KUKA KRL program: ps_604c1.src, ps_604c1.dat

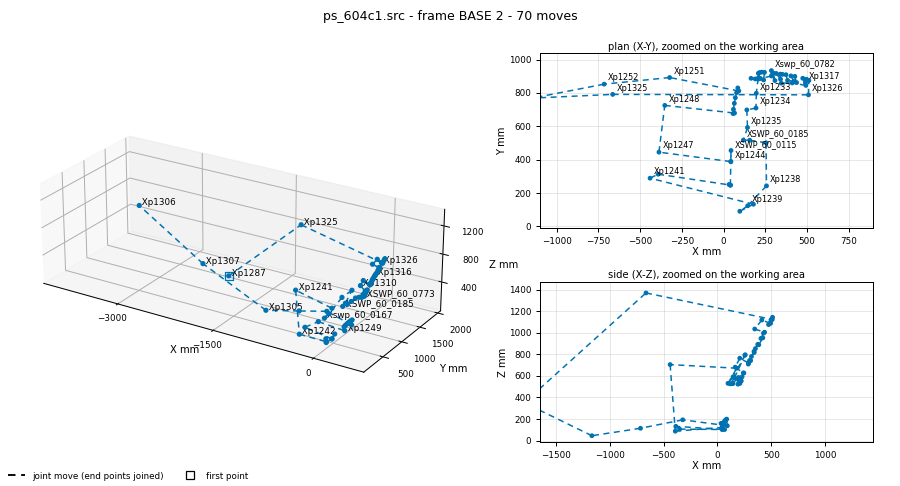
[picture p0: tool path of ps_604c1.src in frame BASE 2, 70 of 70 moves have a stored position in this frame; points joined in program order, loops and branches not executed]
--- ps_604c1.src ---
&ACCESS RVO2
&REL 166
&COMMENT Geom C1 Accelo Atual sem o PTO 60-0682
DEF ps_604c1( )
EXT e_Fraes1 ( )
EXT f_Fraes1 ( )
  ;FOLD INI;%{PE}%V2.2.2,%MKUKATPBASIS,%CINIT,%VCOMMON,%P
  ;FOLD BAS INI;%{PE}%V2.2.2,%MKUKATPBASIS,%CINIT,%VINIT,%P
  INTERRUPT DECL 3 WHEN $STOPMESS==TRUE DO IR_STOPM ( )
  INTERRUPT ON 3
  BAS (#INITMOV,0 )
  ;ENDFOLD
  ;FOLD A20 INI;%{E}%V2.2.2,%MKUKATPA20,%CINIT,%VINIT,%P
  IF ARC20==TRUE THEN
    A20 (ARC_INI)
    INTERRUPT DECL 6 WHEN $CYCFLAG[3]==FALSE DO A20(TECH_STOP2)
  ENDIF
  ;ENDFOLD
  ;FOLD A10 INI;%{E}%V2.2.2,%MKUKATPARC,%CINIT,%VINIT,%P
  IF A10_OPTION==#ACTIVE THEN
    INTERRUPT DECL 4 WHEN $CYCFLAG[2]==FALSE DO A10 (#APPL_ERROR)
    INTERRUPT DECL 7 WHEN A_ARC_SWI==#ACTIVE DO A10 (#ARC_SEAM)
    INTERRUPT DECL 5 WHEN A_FLY_ARC==TRUE DO A10 (#HPU_ARC)
    INTERRUPT  ON 5
    A10_INI ( )
  ENDIF
  ;ENDFOLD
  ;FOLD GRIPPER INI;%{E}%V2.2.2,%MKUKATPGRIPPER,%CINIT,%VINIT,%P
  USER_GRP(0,DUMMY,DUMMY,GDEFAULT)
  ;ENDFOLD
  ;FOLD SPOT INI;%{E}%V.2.2,%MKUKATPSPOT,%CINIT,%VINIT,%P
  USERSPOT(#INIT)
  ;ENDFOLD
  ;FOLD TOUCHSENSE INI;%{E}%V2.2.2,%MKUKATPTS,%CINIT,%VINIT,%P
  IF H70_OPTION THEN
    INTERRUPT DECL 15 WHEN $MEAS_PULSE[TOUCH_I[TOUCH_ACTIVE].IN_NR] DO H70 (6,CD0 )
    INTERRUPT DECL 16 WHEN $ZERO_MOVE DO H70 (7,CD0 )
    INTERRUPT DECL 17 WHEN $TECHPAR_C[FG_TOUCH,8]>0.5 DO H70 (8,CD0)
    H70 (1,CD0 )
  ENDIF
  ;ENDFOLD
  ;FOLD USER INI;%{P}%V2.2.2,%MKUKATPUSER,%CINIT,%VINIT,%P
  ;Make your modifications here
  ;ENDFOLD
  ;ENDFOLD

; Caracterização dos meios de produção: P13.060-R4
; Versão atual: 20/07/2013 12:00  Nome: Solda Geometria C1
; Change: Accelo

chk_w1_wechs_ok ( )     ; VERIFICAÇÃO DE FERRAMENTA: C1

;FOLD PTP p1287 CONT Vel= 80 % PDAT118 Tool[1]:GUN C1 Base[2]:Accelo;%{PE}%R 4.1.16,%MKUKATPBASIS,%CMOVE,%VPTP,%P 1:PTP, 2:p1287, 3:C_PTP, 5:80, 7:PDAT118
$BWDSTART = FALSE
PDAT_ACT=PPDAT118
BAS(#PTP_DAT)
FDAT_ACT=Fp1287
BAS(#FRAMES)
BAS(#VEL_PTP,80)
PTP Xp1287 C_PTP
;ENDFOLD

;FOLD OUT 848 'Area de Solda'  State= FALSE ;%{PE}%R 4.1.16,%MKUKATPBASIS,%COUT,%VOUTX,%P 2:848, 3:'Area de Solda', 5:FALSE, 6:
$OUT[848]=FALSE
;ENDFOLD

;FOLD PTP p1325 CONT Vel= 80 % PDAT36 Tool[1]:GUN C1 Base[2]:Accelo;%{PE}%R 4.1.16,%MKUKATPBASIS,%CMOVE,%VPTP,%P 1:PTP, 2:p1325, 3:C_PTP, 5:80, 7:PDAT36
$BWDSTART = FALSE
PDAT_ACT=PPDAT36
BAS(#PTP_DAT)
FDAT_ACT=Fp1325
BAS(#FRAMES)
BAS(#VEL_PTP,80)
PTP Xp1325 C_PTP
;ENDFOLD
;FOLD PTP p1326 CONT Vel= 80 % PDAT37 Tool[1]:GUN C1 Base[2]:Accelo;%{PE}%R 4.1.16,%MKUKATPBASIS,%CMOVE,%VPTP,%P 1:PTP, 2:p1326, 3:C_PTP, 5:80, 7:PDAT37
$BWDSTART = FALSE
PDAT_ACT=PPDAT37
BAS(#PTP_DAT)
FDAT_ACT=Fp1326
BAS(#FRAMES)
BAS(#VEL_PTP,80)
PTP Xp1326 C_PTP
;ENDFOLD


;FOLD OUT 839 'R4 Soldando'  State= TRUE ;%{PE}%R 4.1.16,%MKUKATPBASIS,%COUT,%VOUTX,%P 2:839, 3:'R4 Soldando', 5:TRUE, 6:
$OUT[839]=TRUE
;ENDFOLD

;FOLD ;  SWP_60_0806;%{PE}%R 4.1.16,%MKUKATPBASIS,%CCOMMENT,%VNORMAL,%P 2: SWP_60_0806
;ENDFOLD
;FOLD PTP swp_60_0806 PDAT38 SPOT Gun= 1 RETR OPN PgNo1= 16 ACTIVE= 1 Tool[1]:GUN C1 Base[2]:Accelo;%{PE}%R 4.1.12,%MKUKATPSPOT,%CSPOT,%VPTP,%P 1:PTP, 2:swp_60_0806, 3:, 5:100, 7:PDAT38, 10:1, 12:#FIRST, 14:#OPN, 16:16, 18:1, 20:0, 22:0, 24:1, 25:NORMAL8
$BWDSTART = FALSE
PDAT_ACT=PPDAT38
BAS(#PTP_DAT)
FDAT_ACT=Fswp_60_0806
BAS(#FRAMES)
BAS(#VEL_PTP,PPDAT38.VEL)
S_ACT.GUN=1
S_ACT.PAIR=SDEFAULT.PAIR
S_ACT.RETR=#OPN
S_ACT.CLO_TM=1
S_ACT.PGNO1=16
S_ACT.PGNO2=SDEFAULT.PGNO2
S_ACT.PRESS1=SDEFAULT.PRESS1
S_ACT.PRESS2=SDEFAULT.PRESS2
S_READY=FALSE
PTP Xswp_60_0806
USERSPOT(#SPOT, S_ACT)
WAIT FOR S_READY
;ENDFOLD

;FOLD ;  SWP_60_0804;%{PE}%R 4.1.16,%MKUKATPBASIS,%CCOMMENT,%VNORMAL,%P 2: SWP_60_0804
;ENDFOLD
;FOLD PTP swp_60_0804 PDAT39 SPOT Gun= 1 RETR OPN PgNo1= 17 ACTIVE= 1 Tool[1]:GUN C1 Base[2]:Accelo;%{PE}%R 4.1.12,%MKUKATPSPOT,%CSPOT,%VPTP,%P 1:PTP, 2:swp_60_0804, 3:, 5:100, 7:PDAT39, 10:1, 12:#FIRST, 14:#OPN, 16:17, 18:1, 20:0, 22:0, 24:1, 25:NORMAL9
$BWDSTART = FALSE
PDAT_ACT=PPDAT39
BAS(#PTP_DAT)
FDAT_ACT=Fswp_60_0804
BAS(#FRAMES)
BAS(#VEL_PTP,PPDAT39.VEL)
S_ACT.GUN=1
S_ACT.PAIR=SDEFAULT.PAIR
S_ACT.RETR=#OPN
S_ACT.CLO_TM=1
S_ACT.PGNO1=17
S_ACT.PGNO2=SDEFAULT.PGNO2
S_ACT.PRESS1=SDEFAULT.PRESS1
S_ACT.PRESS2=SDEFAULT.PRESS2
S_READY=FALSE
PTP Xswp_60_0804
USERSPOT(#SPOT, S_ACT)
WAIT FOR S_READY
;ENDFOLD

;FOLD PTP p1317 CONT Vel= 70 % PDAT40 Tool[1]:GUN C1 Base[2]:Accelo;%{PE}%R 4.1.16,%MKUKATPBASIS,%CMOVE,%VPTP,%P 1:PTP, 2:p1317, 3:C_PTP, 5:70, 7:PDAT40
$BWDSTART = FALSE
PDAT_ACT=PPDAT40
BAS(#PTP_DAT)
FDAT_ACT=Fp1317
BAS(#FRAMES)
BAS(#VEL_PTP,70)
PTP Xp1317 C_PTP
;ENDFOLD

;FOLD ;  SWP_60_0802;%{PE}%R 4.1.16,%MKUKATPBASIS,%CCOMMENT,%VNORMAL,%P 2: SWP_60_0802
;ENDFOLD
;FOLD PTP swp_60_0802 PDAT41 SPOT Gun= 1 RETR OPN PgNo1= 18 ACTIVE= 1 Tool[1]:GUN C1 Base[2]:Accelo;%{PE}%R 4.1.12,%MKUKATPSPOT,%CSPOT,%VPTP,%P 1:PTP, 2:swp_60_0802, 3:, 5:100, 7:PDAT41, 10:1, 12:#FIRST, 14:#OPN, 16:18, 18:1, 20:0, 22:0, 24:1, 25:NORMAL10
$BWDSTART = FALSE
PDAT_ACT=PPDAT41
BAS(#PTP_DAT)
FDAT_ACT=Fswp_60_0802
BAS(#FRAMES)
BAS(#VEL_PTP,PPDAT41.VEL)
S_ACT.GUN=1
S_ACT.PAIR=SDEFAULT.PAIR
S_ACT.RETR=#OPN
S_ACT.CLO_TM=1
S_ACT.PGNO1=18
S_ACT.PGNO2=SDEFAULT.PGNO2
S_ACT.PRESS1=SDEFAULT.PRESS1
S_ACT.PRESS2=SDEFAULT.PRESS2
S_READY=FALSE
PTP Xswp_60_0802
USERSPOT(#SPOT, S_ACT)
WAIT FOR S_READY
;ENDFOLD

;FOLD PTP p1226 CONT Vel= 100 % PDAT57 Tool[1]:GUN C1 Base[2]:Accelo;%{PE}%R 4.1.16,%MKUKATPBASIS,%CMOVE,%VPTP,%P 1:PTP, 2:p1226, 3:C_PTP, 5:100, 7:PDAT57
$BWDSTART = FALSE
PDAT_ACT=PPDAT57
BAS(#PTP_DAT)
FDAT_ACT=Fp1226
BAS(#FRAMES)
BAS(#VEL_PTP,100)
PTP Xp1226 C_PTP
;ENDFOLD
;FOLD PTP p1227 CONT Vel= 100 % PDAT58 Tool[1]:GUN C1 Base[2]:Accelo;%{PE}%R 4.1.16,%MKUKATPBASIS,%CMOVE,%VPTP,%P 1:PTP, 2:p1227, 3:C_PTP, 5:100, 7:PDAT58
$BWDSTART = FALSE
PDAT_ACT=PPDAT58
BAS(#PTP_DAT)
FDAT_ACT=Fp1227
BAS(#FRAMES)
BAS(#VEL_PTP,100)
PTP Xp1227 C_PTP
;ENDFOLD
;FOLD PTP p1228 CONT Vel= 100 % PDAT59 Tool[1]:GUN C1 Base[2]:Accelo;%{PE}%R 4.1.16,%MKUKATPBASIS,%CMOVE,%VPTP,%P 1:PTP, 2:p1228, 3:C_PTP, 5:100, 7:PDAT59
$BWDSTART = FALSE
PDAT_ACT=PPDAT59
BAS(#PTP_DAT)
FDAT_ACT=Fp1228
BAS(#FRAMES)
BAS(#VEL_PTP,100)
PTP Xp1228 C_PTP
;ENDFOLD
;FOLD PTP p1229 CONT Vel= 100 % PDAT60 Tool[1]:GUN C1 Base[2]:Accelo;%{PE}%R 4.1.16,%MKUKATPBASIS,%CMOVE,%VPTP,%P 1:PTP, 2:p1229, 3:C_PTP, 5:100, 7:PDAT60
$BWDSTART = FALSE
PDAT_ACT=PPDAT60
BAS(#PTP_DAT)
FDAT_ACT=Fp1229
BAS(#FRAMES)
BAS(#VEL_PTP,100)
PTP Xp1229 C_PTP
;ENDFOLD

;FOLD ;  SWP_60_0798;%{PE}%R 4.1.16,%MKUKATPBASIS,%CCOMMENT,%VNORMAL,%P 2: SWP_60_0798
;ENDFOLD
;FOLD PTP swp_60_0798 PDAT43 SPOT Gun= 1 RETR OPN PgNo1= 20 ACTIVE= 1 Tool[1]:GUN C1 Base[2]:Accelo;%{PE}%R 4.1.12,%MKUKATPSPOT,%CSPOT,%VPTP,%P 1:PTP, 2:swp_60_0798, 3:, 5:100, 7:PDAT43, 10:1, 12:#FIRST, 14:#OPN, 16:20, 18:1, 20:0, 22:0, 24:1, 25:NORMAL12
$BWDSTART = FALSE
PDAT_ACT=PPDAT43
BAS(#PTP_DAT)
FDAT_ACT=Fswp_60_0798
BAS(#FRAMES)
BAS(#VEL_PTP,PPDAT43.VEL)
S_ACT.GUN=1
S_ACT.PAIR=SDEFAULT.PAIR
S_ACT.RETR=#OPN
S_ACT.CLO_TM=1
S_ACT.PGNO1=20
S_ACT.PGNO2=SDEFAULT.PGNO2
S_ACT.PRESS1=SDEFAULT.PRESS1
S_ACT.PRESS2=SDEFAULT.PRESS2
S_READY=FALSE
PTP Xswp_60_0798
USERSPOT(#SPOT, S_ACT)
WAIT FOR S_READY
;ENDFOLD

;FOLD ;  SWP_60_0794;%{PE}%R 4.1.16,%MKUKATPBASIS,%CCOMMENT,%VNORMAL,%P 2: SWP_60_0794
;ENDFOLD
;FOLD PTP swp_60_0794 PDAT44 SPOT Gun= 1 RETR OPN PgNo1= 21 ACTIVE= 1 Tool[1]:GUN C1 Base[2]:Accelo;%{PE}%R 4.1.12,%MKUKATPSPOT,%CSPOT,%VPTP,%P 1:PTP, 2:swp_60_0794, 3:, 5:100, 7:PDAT44, 10:1, 12:#FIRST, 14:#OPN, 16:21, 18:1, 20:0, 22:0, 24:1, 25:NORMAL13
$BWDSTART = FALSE
PDAT_ACT=PPDAT44
BAS(#PTP_DAT)
FDAT_ACT=Fswp_60_0794
BAS(#FRAMES)
BAS(#VEL_PTP,PPDAT44.VEL)
S_ACT.GUN=1
S_ACT.PAIR=SDEFAULT.PAIR
S_ACT.RETR=#OPN
S_ACT.CLO_TM=1
S_ACT.PGNO1=21
S_ACT.PGNO2=SDEFAULT.PGNO2
S_ACT.PRESS1=SDEFAULT.PRESS1
S_ACT.PRESS2=SDEFAULT.PRESS2
S_READY=FALSE
PTP Xswp_60_0794
USERSPOT(#SPOT, S_ACT)
WAIT FOR S_READY
;ENDFOLD

;FOLD PTP p1282 CONT Vel= 80 % P_OLP77 Tool[1]:GUN C1 Base[2]:Accelo;%{PE}%R 4.1.16,%MKUKATPBASIS,%CMOVE,%VPTP,%P 1:PTP, 2:p1282, 3:C_PTP, 5:80, 7:P_OLP77
$BWDSTART = FALSE
PDAT_ACT=PP_OLP77
BAS(#PTP_DAT)
FDAT_ACT=Fp1282
BAS(#FRAMES)
BAS(#VEL_PTP,80)
PTP Xp1282 C_PTP
;ENDFOLD
;FOLD PTP p1316 CONT Vel= 80 % PDAT45 Tool[1]:GUN C1 Base[2]:Accelo;%{PE}%R 4.1.16,%MKUKATPBASIS,%CMOVE,%VPTP,%P 1:PTP, 2:p1316, 3:C_PTP, 5:80, 7:PDAT45
$BWDSTART = FALSE
PDAT_ACT=PPDAT45
BAS(#PTP_DAT)
FDAT_ACT=Fp1316
BAS(#FRAMES)
BAS(#VEL_PTP,80)
PTP Xp1316 C_PTP
;ENDFOLD

;FOLD ;  SWP_60_0792;%{PE}%R 4.1.16,%MKUKATPBASIS,%CCOMMENT,%VNORMAL,%P 2: SWP_60_0792
;ENDFOLD
;FOLD PTP swp_60_0792 PDAT46 SPOT Gun= 1 RETR OPN PgNo1= 22 ACTIVE= 1 Tool[1]:GUN C1 Base[2]:Accelo;%{PE}%R 4.1.12,%MKUKATPSPOT,%CSPOT,%VPTP,%P 1:PTP, 2:swp_60_0792, 3:, 5:100, 7:PDAT46, 10:1, 12:#FIRST, 14:#OPN, 16:22, 18:1, 20:0, 22:0, 24:1, 25:NORMAL14
$BWDSTART = FALSE
PDAT_ACT=PPDAT46
BAS(#PTP_DAT)
FDAT_ACT=Fswp_60_0792
BAS(#FRAMES)
BAS(#VEL_PTP,PPDAT46.VEL)
S_ACT.GUN=1
S_ACT.PAIR=SDEFAULT.PAIR
S_ACT.RETR=#OPN
S_ACT.CLO_TM=1
S_ACT.PGNO1=22
S_ACT.PGNO2=SDEFAULT.PGNO2
S_ACT.PRESS1=SDEFAULT.PRESS1
S_ACT.PRESS2=SDEFAULT.PRESS2
S_READY=FALSE
PTP Xswp_60_0792
USERSPOT(#SPOT, S_ACT)
WAIT FOR S_READY
;ENDFOLD

;FOLD ;  SWP_60_0790;%{PE}%R 4.1.16,%MKUKATPBASIS,%CCOMMENT,%VNORMAL,%P 2: SWP_60_0790
;ENDFOLD
;FOLD PTP swp_60_0790 PDAT47 SPOT Gun= 1 RETR OPN PgNo1= 23 ACTIVE= 1 Tool[1]:GUN C1 Base[2]:Accelo;%{PE}%R 4.1.12,%MKUKATPSPOT,%CSPOT,%VPTP,%P 1:PTP, 2:swp_60_0790, 3:, 5:100, 7:PDAT47, 10:1, 12:#FIRST, 14:#OPN, 16:23, 18:1, 20:0, 22:0, 24:1, 25:NORMAL15
$BWDSTART = FALSE
PDAT_ACT=PPDAT47
BAS(#PTP_DAT)
FDAT_ACT=Fswp_60_0790
BAS(#FRAMES)
BAS(#VEL_PTP,PPDAT47.VEL)
S_ACT.GUN=1
S_ACT.PAIR=SDEFAULT.PAIR
S_ACT.RETR=#OPN
S_ACT.CLO_TM=1
S_ACT.PGNO1=23
S_ACT.PGNO2=SDEFAULT.PGNO2
S_ACT.PRESS1=SDEFAULT.PRESS1
S_ACT.PRESS2=SDEFAULT.PRESS2
S_READY=FALSE
PTP Xswp_60_0790
USERSPOT(#SPOT, S_ACT)
WAIT FOR S_READY
;ENDFOLD

;FOLD ;  SWP_60_0788;%{PE}%R 4.1.16,%MKUKATPBASIS,%CCOMMENT,%VNORMAL,%P 2: SWP_60_0788
;ENDFOLD
;FOLD PTP swp_60_0788 PDAT48 SPOT Gun= 1 RETR OPN PgNo1= 24 ACTIVE= 1 Tool[1]:GUN C1 Base[2]:Accelo;%{PE}%R 4.1.12,%MKUKATPSPOT,%CSPOT,%VPTP,%P 1:PTP, 2:swp_60_0788, 3:, 5:100, 7:PDAT48, 10:1, 12:#FIRST, 14:#OPN, 16:24, 18:1, 20:0, 22:0, 24:1, 25:NORMAL16
$BWDSTART = FALSE
PDAT_ACT=PPDAT48
BAS(#PTP_DAT)
FDAT_ACT=Fswp_60_0788
BAS(#FRAMES)
BAS(#VEL_PTP,PPDAT48.VEL)
S_ACT.GUN=1
S_ACT.PAIR=SDEFAULT.PAIR
S_ACT.RETR=#OPN
S_ACT.CLO_TM=1
S_ACT.PGNO1=24
S_ACT.PGNO2=SDEFAULT.PGNO2
S_ACT.PRESS1=SDEFAULT.PRESS1
S_ACT.PRESS2=SDEFAULT.PRESS2
S_READY=FALSE
PTP Xswp_60_0788
USERSPOT(#SPOT, S_ACT)
WAIT FOR S_READY
;ENDFOLD

;FOLD PTP p1321 CONT Vel= 80 % PDAT49 Tool[1]:GUN C1 Base[2]:Accelo;%{PE}%R 4.1.16,%MKUKATPBASIS,%CMOVE,%VPTP,%P 1:PTP, 2:p1321, 3:C_PTP, 5:80, 7:PDAT49
$BWDSTART = FALSE
PDAT_ACT=PPDAT49
BAS(#PTP_DAT)
FDAT_ACT=Fp1321
BAS(#FRAMES)
BAS(#VEL_PTP,80)
PTP Xp1321 C_PTP
;ENDFOLD

;FOLD ;  SWP_60_0786;%{PE}%R 4.1.16,%MKUKATPBASIS,%CCOMMENT,%VNORMAL,%P 2: SWP_60_0786
;ENDFOLD
;FOLD PTP swp_60_0786 PDAT50 SPOT Gun= 1 RETR OPN PgNo1= 25 ACTIVE= 1 Tool[1]:GUN C1 Base[2]:Accelo;%{PE}%R 4.1.12,%MKUKATPSPOT,%CSPOT,%VPTP,%P 1:PTP, 2:swp_60_0786, 3:, 5:100, 7:PDAT50, 10:1, 12:#FIRST, 14:#OPN, 16:25, 18:1, 20:0, 22:0, 24:1, 25:NORMAL17
$BWDSTART = FALSE
PDAT_ACT=PPDAT50
BAS(#PTP_DAT)
FDAT_ACT=Fswp_60_0786
BAS(#FRAMES)
BAS(#VEL_PTP,PPDAT50.VEL)
S_ACT.GUN=1
S_ACT.PAIR=SDEFAULT.PAIR
S_ACT.RETR=#OPN
S_ACT.CLO_TM=1
S_ACT.PGNO1=25
S_ACT.PGNO2=SDEFAULT.PGNO2
S_ACT.PRESS1=SDEFAULT.PRESS1
S_ACT.PRESS2=SDEFAULT.PRESS2
S_READY=FALSE
PTP Xswp_60_0786
USERSPOT(#SPOT, S_ACT)
WAIT FOR S_READY
;ENDFOLD

;FOLD ;  SWP_60_0784;%{PE}%R 4.1.16,%MKUKATPBASIS,%CCOMMENT,%VNORMAL,%P 2: SWP_60_0784
;ENDFOLD
;FOLD PTP SWP_60_0785 PDAT117 SPOT Gun= 1 RETR OPN PgNo1= 5 ACTIVE= 1 Tool[1]:GUN C1 Base[2]:Accelo;%{PE}%R 4.1.12,%MKUKATPSPOT,%CSPOT,%VPTP,%P 1:PTP, 2:SWP_60_0785, 3:, 5:100, 7:PDAT117, 10:1, 12:#FIRST, 14:#OPN, 16:5, 18:1, 20:0, 22:0, 24:1, 25:NORMAL22
$BWDSTART = FALSE
PDAT_ACT=PPDAT117
BAS(#PTP_DAT)
FDAT_ACT=FSWP_60_0785
BAS(#FRAMES)
BAS(#VEL_PTP,PPDAT117.VEL)
S_ACT.GUN=1
S_ACT.PAIR=SDEFAULT.PAIR
S_ACT.RETR=#OPN
S_ACT.CLO_TM=1
S_ACT.PGNO1=5
S_ACT.PGNO2=SDEFAULT.PGNO2
S_ACT.PRESS1=SDEFAULT.PRESS1
S_ACT.PRESS2=SDEFAULT.PRESS2
S_READY=FALSE
PTP XSWP_60_0785
USERSPOT(#SPOT, S_ACT)
WAIT FOR S_READY
;ENDFOLD

;FOLD PTP p1322 CONT Vel= 100 % PDAT51 Tool[1]:GUN C1 Base[2]:Accelo;%{PE}%R 4.1.16,%MKUKATPBASIS,%CMOVE,%VPTP,%P 1:PTP, 2:p1322, 3:C_PTP, 5:100, 7:PDAT51
$BWDSTART = FALSE
PDAT_ACT=PPDAT51
BAS(#PTP_DAT)
FDAT_ACT=Fp1322
BAS(#FRAMES)
BAS(#VEL_PTP,100)
PTP Xp1322 C_PTP
;ENDFOLD
;FOLD PTP p1323 CONT Vel= 100 % PDAT52 Tool[1]:GUN C1 Base[2]:Accelo;%{PE}%R 4.1.16,%MKUKATPBASIS,%CMOVE,%VPTP,%P 1:PTP, 2:p1323, 3:C_PTP, 5:100, 7:PDAT52
$BWDSTART = FALSE
PDAT_ACT=PPDAT52
BAS(#PTP_DAT)
FDAT_ACT=Fp1323
BAS(#FRAMES)
BAS(#VEL_PTP,100)
PTP Xp1323 C_PTP
;ENDFOLD

;FOLD ;  SWP_60_0782;%{PE}%R 4.1.16,%MKUKATPBASIS,%CCOMMENT,%VNORMAL,%P 2: SWP_60_0782
;ENDFOLD
;FOLD PTP swp_60_0782 PDAT53 SPOT Gun= 1 RETR OPN PgNo1= 26 ACTIVE= 1 Tool[1]:GUN C1 Base[2]:Accelo;%{PE}%R 4.1.12,%MKUKATPSPOT,%CSPOT,%VPTP,%P 1:PTP, 2:swp_60_0782, 3:, 5:100, 7:PDAT53, 10:1, 12:#FIRST, 14:#OPN, 16:26, 18:1, 20:0, 22:0, 24:1, 25:NORMAL18
$BWDSTART = FALSE
PDAT_ACT=PPDAT53
BAS(#PTP_DAT)
FDAT_ACT=Fswp_60_0782
BAS(#FRAMES)
BAS(#VEL_PTP,PPDAT53.VEL)
S_ACT.GUN=1
S_ACT.PAIR=SDEFAULT.PAIR
S_ACT.RETR=#OPN
S_ACT.CLO_TM=1
S_ACT.PGNO1=26
S_ACT.PGNO2=SDEFAULT.PGNO2
S_ACT.PRESS1=SDEFAULT.PRESS1
S_ACT.PRESS2=SDEFAULT.PRESS2
S_READY=FALSE
PTP Xswp_60_0782
USERSPOT(#SPOT, S_ACT)
WAIT FOR S_READY
;ENDFOLD

;FOLD PTP p1327 CONT Vel= 80 % PDAT55 Tool[1]:GUN C1 Base[2]:Accelo;%{PE}%R 4.1.16,%MKUKATPBASIS,%CMOVE,%VPTP,%P 1:PTP, 2:p1327, 3:C_PTP, 5:80, 7:PDAT55
$BWDSTART = FALSE
PDAT_ACT=PPDAT55
BAS(#PTP_DAT)
FDAT_ACT=Fp1327
BAS(#FRAMES)
BAS(#VEL_PTP,80)
PTP Xp1327 C_PTP
;ENDFOLD
;FOLD PTP p1328 CONT Vel= 80 % PDAT56 Tool[1]:GUN C1 Base[2]:Accelo;%{PE}%R 4.1.16,%MKUKATPBASIS,%CMOVE,%VPTP,%P 1:PTP, 2:p1328, 3:C_PTP, 5:80, 7:PDAT56
$BWDSTART = FALSE
PDAT_ACT=PPDAT56
BAS(#PTP_DAT)
FDAT_ACT=Fp1328
BAS(#FRAMES)
BAS(#VEL_PTP,80)
PTP Xp1328 C_PTP
;ENDFOLD
;FOLD PTP p1310 CONT Vel= 90 % P_OLP78 Tool[1]:GUN C1 Base[2]:Accelo;%{PE}%R 4.1.16,%MKUKATPBASIS,%CMOVE,%VPTP,%P 1:PTP, 2:p1310, 3:C_PTP, 5:90, 7:P_OLP78
$BWDSTART = FALSE
PDAT_ACT=PP_OLP78
BAS(#PTP_DAT)
FDAT_ACT=Fp1310
BAS(#FRAMES)
BAS(#VEL_PTP,90)
PTP Xp1310 C_PTP
;ENDFOLD
;FOLD PTP p1231 CONT Vel= 80 % PDAT62 Tool[1]:GUN C1 Base[2]:Accelo;%{PE}%R 4.1.16,%MKUKATPBASIS,%CMOVE,%VPTP,%P 1:PTP, 2:p1231, 3:C_PTP, 5:80, 7:PDAT62
$BWDSTART = FALSE
PDAT_ACT=PPDAT62
BAS(#PTP_DAT)
FDAT_ACT=Fp1231
BAS(#FRAMES)
BAS(#VEL_PTP,80)
PTP Xp1231 C_PTP
;ENDFOLD

;FOLD ;  SWP_60_0778;%{PE}%R 4.1.16,%MKUKATPBASIS,%CCOMMENT,%VNORMAL,%P 2: SWP_60_0778
;ENDFOLD
;FOLD PTP swp_60_0779 PDAT63 SPOT Gun= 1 RETR OPN PgNo1= 28 ACTIVE= 1 Tool[1]:GUN C1 Base[2]:Accelo;%{PE}%R 4.1.12,%MKUKATPSPOT,%CSPOT,%VPTP,%P 1:PTP, 2:swp_60_0779, 3:, 5:100, 7:PDAT63, 10:1, 12:#FIRST, 14:#OPN, 16:28, 18:1, 20:0, 22:0, 24:1, 25:NORMAL20
$BWDSTART = FALSE
PDAT_ACT=PPDAT63
BAS(#PTP_DAT)
FDAT_ACT=Fswp_60_0779
BAS(#FRAMES)
BAS(#VEL_PTP,PPDAT63.VEL)
S_ACT.GUN=1
S_ACT.PAIR=SDEFAULT.PAIR
S_ACT.RETR=#OPN
S_ACT.CLO_TM=1
S_ACT.PGNO1=28
S_ACT.PGNO2=SDEFAULT.PGNO2
S_ACT.PRESS1=SDEFAULT.PRESS1
S_ACT.PRESS2=SDEFAULT.PRESS2
S_READY=FALSE
PTP Xswp_60_0779
USERSPOT(#SPOT, S_ACT)
WAIT FOR S_READY
;ENDFOLD

;FOLD ;  SWP_60_0776;%{PE}%R 4.1.16,%MKUKATPBASIS,%CCOMMENT,%VNORMAL,%P 2: SWP_60_0776
;ENDFOLD
;FOLD PTP swp_60_0777 PDAT64 SPOT Gun= 1 RETR OPN PgNo1= 29 ACTIVE= 1 Tool[1]:GUN C1 Base[2]:Accelo;%{PE}%R 4.1.12,%MKUKATPSPOT,%CSPOT,%VPTP,%P 1:PTP, 2:swp_60_0777, 3:, 5:100, 7:PDAT64, 10:1, 12:#FIRST, 14:#OPN, 16:29, 18:1, 20:0, 22:0, 24:1, 25:NORMAL20
$BWDSTART = FALSE
PDAT_ACT=PPDAT64
BAS(#PTP_DAT)
FDAT_ACT=Fswp_60_0777
BAS(#FRAMES)
BAS(#VEL_PTP,PPDAT64.VEL)
S_ACT.GUN=1
S_ACT.PAIR=SDEFAULT.PAIR
S_ACT.RETR=#OPN
S_ACT.CLO_TM=1
S_ACT.PGNO1=29
S_ACT.PGNO2=SDEFAULT.PGNO2
S_ACT.PRESS1=SDEFAULT.PRESS1
S_ACT.PRESS2=SDEFAULT.PRESS2
S_READY=FALSE
PTP Xswp_60_0777
USERSPOT(#SPOT, S_ACT)
WAIT FOR S_READY
;ENDFOLD

;FOLD ;  SWP_60_0774;%{PE}%R 4.1.16,%MKUKATPBASIS,%CCOMMENT,%VNORMAL,%P 2: SWP_60_0774
;ENDFOLD
;FOLD PTP swp_60_0775 PDAT65 SPOT Gun= 1 RETR OPN PgNo1= 30 ACTIVE= 1 Tool[1]:GUN C1 Base[2]:Accelo;%{PE}%R 4.1.12,%MKUKATPSPOT,%CSPOT,%VPTP,%P 1:PTP, 2:swp_60_0775, 3:, 5:100, 7:PDAT65, 10:1, 12:#FIRST, 14:#OPN, 16:30, 18:1, 20:0, 22:0, 24:1, 25:NORMAL20
$BWDSTART = FALSE
PDAT_ACT=PPDAT65
BAS(#PTP_DAT)
FDAT_ACT=Fswp_60_0775
BAS(#FRAMES)
BAS(#VEL_PTP,PPDAT65.VEL)
S_ACT.GUN=1
S_ACT.PAIR=SDEFAULT.PAIR
S_ACT.RETR=#OPN
S_ACT.CLO_TM=1
S_ACT.PGNO1=30
S_ACT.PGNO2=SDEFAULT.PGNO2
S_ACT.PRESS1=SDEFAULT.PRESS1
S_ACT.PRESS2=SDEFAULT.PRESS2
S_READY=FALSE
PTP Xswp_60_0775
USERSPOT(#SPOT, S_ACT)
WAIT FOR S_READY
;ENDFOLD
;FOLD PTP p1308 CONT Vel= 80 % PDAT133 Tool[1]:GUN C1 Base[2]:Accelo;%{PE}%R 4.1.16,%MKUKATPBASIS,%CMOVE,%VPTP,%P 1:PTP, 2:p1308, 3:C_PTP, 5:80, 7:PDAT133
$BWDSTART = FALSE
PDAT_ACT=PPDAT133
BAS(#PTP_DAT)
FDAT_ACT=Fp1308
BAS(#FRAMES)
BAS(#VEL_PTP,80)
PTP Xp1308 C_PTP
;ENDFOLD

;FOLD ;  SWP_60_0772;%{PE}%R 4.1.16,%MKUKATPBASIS,%CCOMMENT,%VNORMAL,%P 2: SWP_60_0772
;ENDFOLD
;FOLD PTP SWP_60_0773 PDAT66 SPOT Gun= 1 RETR OPN PgNo1= 4 ACTIVE= 1 Tool[1]:GUN C1 Base[2]:Accelo;%{PE}%R 4.1.12,%MKUKATPSPOT,%CSPOT,%VPTP,%P 1:PTP, 2:SWP_60_0773, 3:, 5:100, 7:PDAT66, 10:1, 12:#FIRST, 14:#OPN, 16:4, 18:1, 20:0, 22:0, 24:1, 25:NORMAL20
$BWDSTART = FALSE
PDAT_ACT=PPDAT66
BAS(#PTP_DAT)
FDAT_ACT=FSWP_60_0773
BAS(#FRAMES)
BAS(#VEL_PTP,PPDAT66.VEL)
S_ACT.GUN=1
S_ACT.PAIR=SDEFAULT.PAIR
S_ACT.RETR=#OPN
S_ACT.CLO_TM=1
S_ACT.PGNO1=4
S_ACT.PGNO2=SDEFAULT.PGNO2
S_ACT.PRESS1=SDEFAULT.PRESS1
S_ACT.PRESS2=SDEFAULT.PRESS2
S_READY=FALSE
PTP XSWP_60_0773
USERSPOT(#SPOT, S_ACT)
WAIT FOR S_READY
;ENDFOLD

;FOLD PTP p1232 CONT Vel= 90 % P_OLP79 Tool[1]:GUN C1 Base[2]:Accelo;%{PE}%R 4.1.16,%MKUKATPBASIS,%CMOVE,%VPTP,%P 1:PTP, 2:p1232, 3:C_PTP, 5:90, 7:P_OLP79
$BWDSTART = FALSE
PDAT_ACT=PP_OLP79
BAS(#PTP_DAT)
FDAT_ACT=Fp1232
BAS(#FRAMES)
BAS(#VEL_PTP,90)
PTP Xp1232 C_PTP
;ENDFOLD

;FOLD ;  SWP_60_0198;%{PE}%R 4.1.16,%MKUKATPBASIS,%CCOMMENT,%VNORMAL,%P 2: SWP_60_0198
;ENDFOLD
;FOLD PTP SWP_60_0199 PDAT67 SPOT Gun= 1 RETR OPN PgNo1= 3 ACTIVE= 1 Tool[1]:GUN C1 Base[2]:Accelo;%{PE}%R 4.1.12,%MKUKATPSPOT,%CSPOT,%VPTP,%P 1:PTP, 2:SWP_60_0199, 3:, 5:100, 7:PDAT67, 10:1, 12:#FIRST, 14:#OPN, 16:3, 18:1, 20:0, 22:0, 24:1, 25:NORMAL20
$BWDSTART = FALSE
PDAT_ACT=PPDAT67
BAS(#PTP_DAT)
FDAT_ACT=FSWP_60_0199
BAS(#FRAMES)
BAS(#VEL_PTP,PPDAT67.VEL)
S_ACT.GUN=1
S_ACT.PAIR=SDEFAULT.PAIR
S_ACT.RETR=#OPN
S_ACT.CLO_TM=1
S_ACT.PGNO1=3
S_ACT.PGNO2=SDEFAULT.PGNO2
S_ACT.PRESS1=SDEFAULT.PRESS1
S_ACT.PRESS2=SDEFAULT.PRESS2
S_READY=FALSE
PTP XSWP_60_0199
USERSPOT(#SPOT, S_ACT)
WAIT FOR S_READY
;ENDFOLD

;FOLD PTP p1286 CONT Vel= 80 % PDAT116 Tool[1]:GUN C1 Base[2]:Accelo;%{PE}%R 4.1.16,%MKUKATPBASIS,%CMOVE,%VPTP,%P 1:PTP, 2:p1286, 3:C_PTP, 5:80, 7:PDAT116
$BWDSTART = FALSE
PDAT_ACT=PPDAT116
BAS(#PTP_DAT)
FDAT_ACT=Fp1286
BAS(#FRAMES)
BAS(#VEL_PTP,80)
PTP Xp1286 C_PTP
;ENDFOLD
;FOLD PTP p1233 CONT Vel= 80 % PDAT78 Tool[1]:GUN C1 Base[2]:Accelo;%{PE}%R 4.1.16,%MKUKATPBASIS,%CMOVE,%VPTP,%P 1:PTP, 2:p1233, 3:C_PTP, 5:80, 7:PDAT78
$BWDSTART = FALSE
PDAT_ACT=PPDAT78
BAS(#PTP_DAT)
FDAT_ACT=Fp1233
BAS(#FRAMES)
BAS(#VEL_PTP,80)
PTP Xp1233 C_PTP
;ENDFOLD
;FOLD PTP p1234 CONT Vel= 80 % PDAT79 Tool[1]:GUN C1 Base[2]:Accelo;%{PE}%R 4.1.16,%MKUKATPBASIS,%CMOVE,%VPTP,%P 1:PTP, 2:p1234, 3:C_PTP, 5:80, 7:PDAT79
$BWDSTART = FALSE
PDAT_ACT=PPDAT79
BAS(#PTP_DAT)
FDAT_ACT=Fp1234
BAS(#FRAMES)
BAS(#VEL_PTP,80)
PTP Xp1234 C_PTP
;ENDFOLD

;FOLD ;  SWP_60_0192;%{PE}%R 4.1.16,%MKUKATPBASIS,%CCOMMENT,%VNORMAL,%P 2: SWP_60_0192
;ENDFOLD
;FOLD PTP swp_60_0193 PDAT68 SPOT Gun= 1 RETR OPN PgNo1= 31 ACTIVE= 1 Tool[1]:GUN C1 Base[2]:Accelo;%{PE}%R 4.1.12,%MKUKATPSPOT,%CSPOT,%VPTP,%P 1:PTP, 2:swp_60_0193, 3:, 5:100, 7:PDAT68, 10:1, 12:#FIRST, 14:#OPN, 16:31, 18:1, 20:0, 22:0, 24:1, 25:NORMAL20
$BWDSTART = FALSE
PDAT_ACT=PPDAT68
BAS(#PTP_DAT)
FDAT_ACT=Fswp_60_0193
BAS(#FRAMES)
BAS(#VEL_PTP,PPDAT68.VEL)
S_ACT.GUN=1
S_ACT.PAIR=SDEFAULT.PAIR
S_ACT.RETR=#OPN
S_ACT.CLO_TM=1
S_ACT.PGNO1=31
S_ACT.PGNO2=SDEFAULT.PGNO2
S_ACT.PRESS1=SDEFAULT.PRESS1
S_ACT.PRESS2=SDEFAULT.PRESS2
S_READY=FALSE
PTP Xswp_60_0193
USERSPOT(#SPOT, S_ACT)
WAIT FOR S_READY
;ENDFOLD

;FOLD PTP p1235 CONT Vel= 80 % PDAT80 Tool[1]:GUN C1 Base[2]:Accelo;%{PE}%R 4.1.16,%MKUKATPBASIS,%CMOVE,%VPTP,%P 1:PTP, 2:p1235, 3:C_PTP, 5:80, 7:PDAT80
$BWDSTART = FALSE
PDAT_ACT=PPDAT80
BAS(#PTP_DAT)
FDAT_ACT=Fp1235
BAS(#FRAMES)
BAS(#VEL_PTP,80)
PTP Xp1235 C_PTP
;ENDFOLD

;FOLD ;  SWP_60_0184;%{PE}%R 4.1.16,%MKUKATPBASIS,%CCOMMENT,%VNORMAL,%P 2: SWP_60_0184
;ENDFOLD
;FOLD PTP SWP_60_0185 PDAT69 SPOT Gun= 1 RETR OPN PgNo1= 2 ACTIVE= 1 Tool[1]:GUN C1 Base[2]:Accelo;%{PE}%R 4.1.12,%MKUKATPSPOT,%CSPOT,%VPTP,%P 1:PTP, 2:SWP_60_0185, 3:, 5:100, 7:PDAT69, 10:1, 12:#FIRST, 14:#OPN, 16:2, 18:1, 20:0, 22:0, 24:1, 25:NORMAL20
$BWDSTART = FALSE
PDAT_ACT=PPDAT69
BAS(#PTP_DAT)
FDAT_ACT=FSWP_60_0185
BAS(#FRAMES)
BAS(#VEL_PTP,PPDAT69.VEL)
S_ACT.GUN=1
S_ACT.PAIR=SDEFAULT.PAIR
S_ACT.RETR=#OPN
S_ACT.CLO_TM=1
S_ACT.PGNO1=2
S_ACT.PGNO2=SDEFAULT.PGNO2
S_ACT.PRESS1=SDEFAULT.PRESS1
S_ACT.PRESS2=SDEFAULT.PRESS2
S_READY=FALSE
PTP XSWP_60_0185
USERSPOT(#SPOT, S_ACT)
WAIT FOR S_READY
;ENDFOLD

;FOLD Kollision.Ueberwachung_3_Ein ;%{PE}%MKUKATPUSER
COLLSTOP( 3, 1 ) ;INTERRUPTUEBERWACHT
;ENDFOLD

;FOLD PTP p1236 CONT Vel= 80 % PDAT81 Tool[1]:GUN C1 Base[2]:Accelo;%{PE}%R 4.1.16,%MKUKATPBASIS,%CMOVE,%VPTP,%P 1:PTP, 2:p1236, 3:C_PTP, 5:80, 7:PDAT81
$BWDSTART = FALSE
PDAT_ACT=PPDAT81
BAS(#PTP_DAT)
FDAT_ACT=Fp1236
BAS(#FRAMES)
BAS(#VEL_PTP,80)
PTP Xp1236 C_PTP
;ENDFOLD
;FOLD PTP p1237 CONT Vel= 80 % PDAT82 Tool[1]:GUN C1 Base[2]:Accelo;%{PE}%R 4.1.16,%MKUKATPBASIS,%CMOVE,%VPTP,%P 1:PTP, 2:p1237, 3:C_PTP, 5:80, 7:PDAT82
$BWDSTART = FALSE
PDAT_ACT=PPDAT82
BAS(#PTP_DAT)
FDAT_ACT=Fp1237
BAS(#FRAMES)
BAS(#VEL_PTP,80)
PTP Xp1237 C_PTP
;ENDFOLD
;FOLD PTP p1238 CONT Vel= 80 % PDAT83 Tool[1]:GUN C1 Base[2]:Accelo;%{PE}%R 4.1.16,%MKUKATPBASIS,%CMOVE,%VPTP,%P 1:PTP, 2:p1238, 3:C_PTP, 5:80, 7:PDAT83
$BWDSTART = FALSE
PDAT_ACT=PPDAT83
BAS(#PTP_DAT)
FDAT_ACT=Fp1238
BAS(#FRAMES)
BAS(#VEL_PTP,80)
PTP Xp1238 C_PTP
;ENDFOLD
;FOLD PTP p1239 CONT Vel= 80 % PDAT84 Tool[1]:GUN C1 Base[2]:Accelo;%{PE}%R 4.1.16,%MKUKATPBASIS,%CMOVE,%VPTP,%P 1:PTP, 2:p1239, 3:C_PTP, 5:80, 7:PDAT84
$BWDSTART = FALSE
PDAT_ACT=PPDAT84
BAS(#PTP_DAT)
FDAT_ACT=Fp1239
BAS(#FRAMES)
BAS(#VEL_PTP,80)
PTP Xp1239 C_PTP
;ENDFOLD

;FOLD ;  SWP_60_0166;%{PE}%R 4.1.16,%MKUKATPBASIS,%CCOMMENT,%VNORMAL,%P 2: SWP_60_0166
;ENDFOLD
;FOLD PTP swp_60_0167 PDAT70 SPOT Gun= 1 RETR OPN PgNo1= 1 ACTIVE= 1 Tool[1]:GUN C1 Base[2]:Accelo;%{PE}%R 4.1.12,%MKUKATPSPOT,%CSPOT,%VPTP,%P 1:PTP, 2:swp_60_0167, 3:, 5:100, 7:PDAT70, 10:1, 12:#FIRST, 14:#OPN, 16:1, 18:1, 20:0, 22:0, 24:1, 25:NORMAL20
$BWDSTART = FALSE
PDAT_ACT=PPDAT70
BAS(#PTP_DAT)
FDAT_ACT=Fswp_60_0167
BAS(#FRAMES)
BAS(#VEL_PTP,PPDAT70.VEL)
S_ACT.GUN=1
S_ACT.PAIR=SDEFAULT.PAIR
S_ACT.RETR=#OPN
S_ACT.CLO_TM=1
S_ACT.PGNO1=1
S_ACT.PGNO2=SDEFAULT.PGNO2
S_ACT.PRESS1=SDEFAULT.PRESS1
S_ACT.PRESS2=SDEFAULT.PRESS2
S_READY=FALSE
PTP Xswp_60_0167
USERSPOT(#SPOT, S_ACT)
WAIT FOR S_READY
;ENDFOLD

;FOLD PTP p1240 CONT Vel= 80 % PDAT85 Tool[1]:GUN C1 Base[2]:Accelo;%{PE}%R 4.1.16,%MKUKATPBASIS,%CMOVE,%VPTP,%P 1:PTP, 2:p1240, 3:C_PTP, 5:80, 7:PDAT85
$BWDSTART = FALSE
PDAT_ACT=PPDAT85
BAS(#PTP_DAT)
FDAT_ACT=Fp1240
BAS(#FRAMES)
BAS(#VEL_PTP,80)
PTP Xp1240 C_PTP
;ENDFOLD
;FOLD PTP p1241 CONT Vel= 80 % PDAT86 Tool[1]:GUN C1 Base[2]:Accelo;%{PE}%R 4.1.16,%MKUKATPBASIS,%CMOVE,%VPTP,%P 1:PTP, 2:p1241, 3:C_PTP, 5:80, 7:PDAT86
$BWDSTART = FALSE
PDAT_ACT=PPDAT86
BAS(#PTP_DAT)
FDAT_ACT=Fp1241
BAS(#FRAMES)
BAS(#VEL_PTP,80)
PTP Xp1241 C_PTP
;ENDFOLD
;FOLD PTP p1242 CONT Vel= 80 % PDAT87 Tool[1]:GUN C1 Base[2]:Accelo;%{PE}%R 4.1.16,%MKUKATPBASIS,%CMOVE,%VPTP,%P 1:PTP, 2:p1242, 3:C_PTP, 5:80, 7:PDAT87
$BWDSTART = FALSE
PDAT_ACT=PPDAT87
BAS(#PTP_DAT)
FDAT_ACT=Fp1242
BAS(#FRAMES)
BAS(#VEL_PTP,80)
PTP Xp1242 C_PTP
;ENDFOLD
;FOLD PTP p1243 CONT Vel= 80 % PDAT88 Tool[1]:GUN C1 Base[2]:Accelo;%{PE}%R 4.1.16,%MKUKATPBASIS,%CMOVE,%VPTP,%P 1:PTP, 2:p1243, 3:C_PTP, 5:80, 7:PDAT88
$BWDSTART = FALSE
PDAT_ACT=PPDAT88
BAS(#PTP_DAT)
FDAT_ACT=Fp1243
BAS(#FRAMES)
BAS(#VEL_PTP,80)
PTP Xp1243 C_PTP
;ENDFOLD

;FOLD ;  SWP_60_0102;%{PE}%R 4.1.16,%MKUKATPBASIS,%CCOMMENT,%VNORMAL,%P 2: SWP_60_0102
;ENDFOLD
;FOLD PTP SWP_60_0103 PDAT71 SPOT Gun= 1 RETR OPN PgNo1= 7 ACTIVE= 1 Tool[1]:GUN C1 Base[2]:Accelo;%{PE}%R 4.1.12,%MKUKATPSPOT,%CSPOT,%VPTP,%P 1:PTP, 2:SWP_60_0103, 3:, 5:100, 7:PDAT71, 10:1, 12:#FIRST, 14:#OPN, 16:7, 18:1, 20:0, 22:0, 24:1, 25:NORMAL20
$BWDSTART = FALSE
PDAT_ACT=PPDAT71
BAS(#PTP_DAT)
FDAT_ACT=FSWP_60_0103
BAS(#FRAMES)
BAS(#VEL_PTP,PPDAT71.VEL)
S_ACT.GUN=1
S_ACT.PAIR=SDEFAULT.PAIR
S_ACT.RETR=#OPN
S_ACT.CLO_TM=1
S_ACT.PGNO1=7
S_ACT.PGNO2=SDEFAULT.PGNO2
S_ACT.PRESS1=SDEFAULT.PRESS1
S_ACT.PRESS2=SDEFAULT.PRESS2
S_READY=FALSE
PTP XSWP_60_0103
USERSPOT(#SPOT, S_ACT)
WAIT FOR S_READY
;ENDFOLD

;FOLD PTP p1245 CONT Vel= 80 % PDAT90 Tool[1]:GUN C1 Base[2]:Accelo;%{PE}%R 4.1.16,%MKUKATPBASIS,%CMOVE,%VPTP,%P 1:PTP, 2:p1245, 3:C_PTP, 5:80, 7:PDAT90
$BWDSTART = FALSE
PDAT_ACT=PPDAT90
BAS(#PTP_DAT)
FDAT_ACT=Fp1245
BAS(#FRAMES)
BAS(#VEL_PTP,80)
PTP Xp1245 C_PTP
;ENDFOLD
;FOLD PTP p1244 CONT Vel= 80 % PDAT89 Tool[1]:GUN C1 Base[2]:Accelo;%{PE}%R 4.1.16,%MKUKATPBASIS,%CMOVE,%VPTP,%P 1:PTP, 2:p1244, 3:C_PTP, 5:80, 7:PDAT89
$BWDSTART = FALSE
PDAT_ACT=PPDAT89
BAS(#PTP_DAT)
FDAT_ACT=Fp1244
BAS(#FRAMES)
BAS(#VEL_PTP,80)
PTP Xp1244 C_PTP
;ENDFOLD

;FOLD ;  SWP_60_0114;%{PE}%R 4.1.16,%MKUKATPBASIS,%CCOMMENT,%VNORMAL,%P 2: SWP_60_0114
;ENDFOLD
;FOLD PTP SWP_60_0115 PDAT72 SPOT Gun= 1 RETR OPN PgNo1= 8 ACTIVE= 1 Tool[1]:GUN C1 Base[2]:Accelo;%{PE}%R 4.1.12,%MKUKATPSPOT,%CSPOT,%VPTP,%P 1:PTP, 2:SWP_60_0115, 3:, 5:100, 7:PDAT72, 10:1, 12:#FIRST, 14:#OPN, 16:8, 18:1, 20:0, 22:0, 24:1, 25:NORMAL20
$BWDSTART = FALSE
PDAT_ACT=PPDAT72
BAS(#PTP_DAT)
FDAT_ACT=FSWP_60_0115
BAS(#FRAMES)
BAS(#VEL_PTP,PPDAT72.VEL)
S_ACT.GUN=1
S_ACT.PAIR=SDEFAULT.PAIR
S_ACT.RETR=#OPN
S_ACT.CLO_TM=1
S_ACT.PGNO1=8
S_ACT.PGNO2=SDEFAULT.PGNO2
S_ACT.PRESS1=SDEFAULT.PRESS1
S_ACT.PRESS2=SDEFAULT.PRESS2
S_READY=FALSE
PTP XSWP_60_0115
USERSPOT(#SPOT, S_ACT)
WAIT FOR S_READY
;ENDFOLD

;FOLD PTP p1246 CONT Vel= 80 % PDAT91 Tool[1]:GUN C1 Base[2]:Accelo;%{PE}%R 4.1.16,%MKUKATPBASIS,%CMOVE,%VPTP,%P 1:PTP, 2:p1246, 3:C_PTP, 5:80, 7:PDAT91
$BWDSTART = FALSE
PDAT_ACT=PPDAT91
BAS(#PTP_DAT)
FDAT_ACT=Fp1246
BAS(#FRAMES)
BAS(#VEL_PTP,80)
PTP Xp1246 C_PTP
;ENDFOLD
;FOLD PTP p1247 CONT Vel= 80 % PDAT92 Tool[1]:GUN C1 Base[2]:Accelo;%{PE}%R 4.1.16,%MKUKATPBASIS,%CMOVE,%VPTP,%P 1:PTP, 2:p1247, 3:C_PTP, 5:80, 7:PDAT92
$BWDSTART = FALSE
PDAT_ACT=PPDAT92
BAS(#PTP_DAT)
FDAT_ACT=Fp1247
BAS(#FRAMES)
BAS(#VEL_PTP,80)
PTP Xp1247 C_PTP
;ENDFOLD
;FOLD PTP p1248 CONT Vel= 80 % PDAT93 Tool[1]:GUN C1 Base[2]:Accelo;%{PE}%R 4.1.16,%MKUKATPBASIS,%CMOVE,%VPTP,%P 1:PTP, 2:p1248, 3:C_PTP, 5:80, 7:PDAT93
$BWDSTART = FALSE
PDAT_ACT=PPDAT93
BAS(#PTP_DAT)
FDAT_ACT=Fp1248
BAS(#FRAMES)
BAS(#VEL_PTP,80)
PTP Xp1248 C_PTP
;ENDFOLD
;FOLD PTP p1249 CONT Vel= 80 % PDAT94 Tool[1]:GUN C1 Base[2]:Accelo;%{PE}%R 4.1.16,%MKUKATPBASIS,%CMOVE,%VPTP,%P 1:PTP, 2:p1249, 3:C_PTP, 5:80, 7:PDAT94
$BWDSTART = FALSE
PDAT_ACT=PPDAT94
BAS(#PTP_DAT)
FDAT_ACT=Fp1249
BAS(#FRAMES)
BAS(#VEL_PTP,80)
PTP Xp1249 C_PTP
;ENDFOLD

;FOLD Kollision.Ueberwachung_3_Aus ;%{PE}%MKUKATPUSER
COLLSTOP( 3, 2 )
;ENDFOLD

;FOLD ;  SWP_60_0116;%{PE}%R 4.1.16,%MKUKATPBASIS,%CCOMMENT,%VNORMAL,%P 2: SWP_60_0116
;ENDFOLD
;FOLD PTP SWP_60_0117 PDAT73 SPOT Gun= 1 RETR OPN PgNo1= 9 ACTIVE= 1 Tool[1]:GUN C1 Base[2]:Accelo;%{PE}%R 4.1.12,%MKUKATPSPOT,%CSPOT,%VPTP,%P 1:PTP, 2:SWP_60_0117, 3:, 5:100, 7:PDAT73, 10:1, 12:#FIRST, 14:#OPN, 16:9, 18:1, 20:0, 22:0, 24:1, 25:NORMAL20
$BWDSTART = FALSE
PDAT_ACT=PPDAT73
BAS(#PTP_DAT)
FDAT_ACT=FSWP_60_0117
BAS(#FRAMES)
BAS(#VEL_PTP,PPDAT73.VEL)
S_ACT.GUN=1
S_ACT.PAIR=SDEFAULT.PAIR
S_ACT.RETR=#OPN
S_ACT.CLO_TM=1
S_ACT.PGNO1=9
S_ACT.PGNO2=SDEFAULT.PGNO2
S_ACT.PRESS1=SDEFAULT.PRESS1
S_ACT.PRESS2=SDEFAULT.PRESS2
S_READY=FALSE
PTP XSWP_60_0117
USERSPOT(#SPOT, S_ACT)
WAIT FOR S_READY
;ENDFOLD

;FOLD ;  SWP_60_0118;%{PE}%R 4.1.16,%MKUKATPBASIS,%CCOMMENT,%VNORMAL,%P 2: SWP_60_0118
;ENDFOLD
;FOLD PTP swp_60_0119 PDAT74 SPOT Gun= 1 RETR OPN PgNo1= 32 ACTIVE= 1 Tool[1]:GUN C1 Base[2]:Accelo;%{PE}%R 4.1.12,%MKUKATPSPOT,%CSPOT,%VPTP,%P 1:PTP, 2:swp_60_0119, 3:, 5:100, 7:PDAT74, 10:1, 12:#FIRST, 14:#OPN, 16:32, 18:1, 20:0, 22:0, 24:1, 25:NORMAL20
$BWDSTART = FALSE
PDAT_ACT=PPDAT74
BAS(#PTP_DAT)
FDAT_ACT=Fswp_60_0119
BAS(#FRAMES)
BAS(#VEL_PTP,PPDAT74.VEL)
S_ACT.GUN=1
S_ACT.PAIR=SDEFAULT.PAIR
S_ACT.RETR=#OPN
S_ACT.CLO_TM=1
S_ACT.PGNO1=32
S_ACT.PGNO2=SDEFAULT.PGNO2
S_ACT.PRESS1=SDEFAULT.PRESS1
S_ACT.PRESS2=SDEFAULT.PRESS2
S_READY=FALSE
PTP Xswp_60_0119
USERSPOT(#SPOT, S_ACT)
WAIT FOR S_READY
;ENDFOLD

;FOLD ;  SWP_60_0120;%{PE}%R 4.1.16,%MKUKATPBASIS,%CCOMMENT,%VNORMAL,%P 2: SWP_60_0120
;ENDFOLD
;FOLD PTP swp_60_0121 PDAT75 SPOT Gun= 1 RETR OPN PgNo1= 33 ACTIVE= 1 Tool[1]:GUN C1 Base[2]:Accelo;%{PE}%R 4.1.12,%MKUKATPSPOT,%CSPOT,%VPTP,%P 1:PTP, 2:swp_60_0121, 3:, 5:100, 7:PDAT75, 10:1, 12:#FIRST, 14:#OPN, 16:33, 18:1, 20:0, 22:0, 24:1, 25:NORMAL20
$BWDSTART = FALSE
PDAT_ACT=PPDAT75
BAS(#PTP_DAT)
FDAT_ACT=Fswp_60_0121
BAS(#FRAMES)
BAS(#VEL_PTP,PPDAT75.VEL)
S_ACT.GUN=1
S_ACT.PAIR=SDEFAULT.PAIR
S_ACT.RETR=#OPN
S_ACT.CLO_TM=1
S_ACT.PGNO1=33
S_ACT.PGNO2=SDEFAULT.PGNO2
S_ACT.PRESS1=SDEFAULT.PRESS1
S_ACT.PRESS2=SDEFAULT.PRESS2
S_READY=FALSE
PTP Xswp_60_0121
USERSPOT(#SPOT, S_ACT)
WAIT FOR S_READY
;ENDFOLD

;FOLD ;  SWP_60_0122;%{PE}%R 4.1.16,%MKUKATPBASIS,%CCOMMENT,%VNORMAL,%P 2: SWP_60_0122
;ENDFOLD
;FOLD PTP swp_60_0123 PDAT76 SPOT Gun= 1 RETR OPN PgNo1= 34 ACTIVE= 1 Tool[1]:GUN C1 Base[2]:Accelo;%{PE}%R 4.1.12,%MKUKATPSPOT,%CSPOT,%VPTP,%P 1:PTP, 2:swp_60_0123, 3:, 5:100, 7:PDAT76, 10:1, 12:#FIRST, 14:#OPN, 16:34, 18:1, 20:0, 22:0, 24:1, 25:NORMAL20
$BWDSTART = FALSE
PDAT_ACT=PPDAT76
BAS(#PTP_DAT)
FDAT_ACT=Fswp_60_0123
BAS(#FRAMES)
BAS(#VEL_PTP,PPDAT76.VEL)
S_ACT.GUN=1
S_ACT.PAIR=SDEFAULT.PAIR
S_ACT.RETR=#OPN
S_ACT.CLO_TM=1
S_ACT.PGNO1=34
S_ACT.PGNO2=SDEFAULT.PGNO2
S_ACT.PRESS1=SDEFAULT.PRESS1
S_ACT.PRESS2=SDEFAULT.PRESS2
S_READY=FALSE
PTP Xswp_60_0123
USERSPOT(#SPOT, S_ACT)
WAIT FOR S_READY
;ENDFOLD

;FOLD ;  SWP_60_0124;%{PE}%R 4.1.16,%MKUKATPBASIS,%CCOMMENT,%VNORMAL,%P 2: SWP_60_0124
;ENDFOLD
;FOLD PTP swp_60_0125 PDAT95 SPOT Gun= 1 RETR OPN PgNo1= 35 ACTIVE= 1 Tool[1]:GUN C1 Base[2]:Accelo;%{PE}%R 4.1.12,%MKUKATPSPOT,%CSPOT,%VPTP,%P 1:PTP, 2:swp_60_0125, 3:, 5:100, 7:PDAT95, 10:1, 12:#FIRST, 14:#OPN, 16:35, 18:1, 20:0, 22:0, 24:1, 25:NORMAL20
$BWDSTART = FALSE
PDAT_ACT=PPDAT95
BAS(#PTP_DAT)
FDAT_ACT=Fswp_60_0125
BAS(#FRAMES)
BAS(#VEL_PTP,PPDAT95.VEL)
S_ACT.GUN=1
S_ACT.PAIR=SDEFAULT.PAIR
S_ACT.RETR=#OPN
S_ACT.CLO_TM=1
S_ACT.PGNO1=35
S_ACT.PGNO2=SDEFAULT.PGNO2
S_ACT.PRESS1=SDEFAULT.PRESS1
S_ACT.PRESS2=SDEFAULT.PRESS2
S_READY=FALSE
PTP Xswp_60_0125
USERSPOT(#SPOT, S_ACT)
WAIT FOR S_READY
;ENDFOLD

;FOLD ;  SWP_60_0126;%{PE}%R 4.1.16,%MKUKATPBASIS,%CCOMMENT,%VNORMAL,%P 2: SWP_60_0126
;ENDFOLD
;FOLD PTP SWP_60_0127 PDAT77 SPOT Gun= 1 RETR OPN PgNo1= 10 ACTIVE= 1 Tool[1]:GUN C1 Base[2]:Accelo;%{PE}%R 4.1.12,%MKUKATPSPOT,%CSPOT,%VPTP,%P 1:PTP, 2:SWP_60_0127, 3:, 5:100, 7:PDAT77, 10:1, 12:#FIRST, 14:#OPN, 16:10, 18:1, 20:0, 22:0, 24:1, 25:NORMAL20
$BWDSTART = FALSE
PDAT_ACT=PPDAT77
BAS(#PTP_DAT)
FDAT_ACT=FSWP_60_0127
BAS(#FRAMES)
BAS(#VEL_PTP,PPDAT77.VEL)
S_ACT.GUN=1
S_ACT.PAIR=SDEFAULT.PAIR
S_ACT.RETR=#OPN
S_ACT.CLO_TM=1
S_ACT.PGNO1=10
S_ACT.PGNO2=SDEFAULT.PGNO2
S_ACT.PRESS1=SDEFAULT.PRESS1
S_ACT.PRESS2=SDEFAULT.PRESS2
S_READY=FALSE
PTP XSWP_60_0127
USERSPOT(#SPOT, S_ACT)
WAIT FOR S_READY
;ENDFOLD

;FOLD PTP p1250 CONT Vel= 80 % PDAT96 Tool[1]:GUN C1 Base[2]:Accelo;%{PE}%R 4.1.16,%MKUKATPBASIS,%CMOVE,%VPTP,%P 1:PTP, 2:p1250, 3:C_PTP, 5:80, 7:PDAT96
$BWDSTART = FALSE
PDAT_ACT=PPDAT96
BAS(#PTP_DAT)
FDAT_ACT=Fp1250
BAS(#FRAMES)
BAS(#VEL_PTP,80)
PTP Xp1250 C_PTP
;ENDFOLD
;FOLD PTP p1251 CONT Vel= 80 % PDAT97 Tool[1]:GUN C1 Base[2]:Accelo;%{PE}%R 4.1.16,%MKUKATPBASIS,%CMOVE,%VPTP,%P 1:PTP, 2:p1251, 3:C_PTP, 5:80, 7:PDAT97
$BWDSTART = FALSE
PDAT_ACT=PPDAT97
BAS(#PTP_DAT)
FDAT_ACT=Fp1251
BAS(#FRAMES)
BAS(#VEL_PTP,80)
PTP Xp1251 C_PTP
;ENDFOLD
;FOLD PTP p1252 CONT Vel= 80 % PDAT98 Tool[1]:GUN C1 Base[2]:Accelo;%{PE}%R 4.1.16,%MKUKATPBASIS,%CMOVE,%VPTP,%P 1:PTP, 2:p1252, 3:C_PTP, 5:80, 7:PDAT98
$BWDSTART = FALSE
PDAT_ACT=PPDAT98
BAS(#PTP_DAT)
FDAT_ACT=Fp1252
BAS(#FRAMES)
BAS(#VEL_PTP,80)
PTP Xp1252 C_PTP
;ENDFOLD

;FOLD ;  SWP_60_0682 Prg Solda 13 foi p/ R2 GEO3;%{PE}%R 4.1.16,%MKUKATPBASIS,%CCOMMENT,%VNORMAL,%P 2: SWP_60_0682 Prg Solda 13 foi p/ R2 GEO3
;ENDFOLD

;FOLD ; Alterado A848 para false;%{PE}%R 4.1.16,%MKUKATPBASIS,%CCOMMENT,%VNORMAL,%P 2:Alterado A848 para false
;ENDFOLD
;FOLD OUT 848 'Area de Solda'  State= FALSE CONT;%{PE}%R 4.1.16,%MKUKATPBASIS,%COUT,%VOUTX,%P 2:848, 3:'Area de Solda', 5:FALSE, 6:CONTINUE
CONTINUE
$OUT[848]=FALSE
;ENDFOLD

;FOLD ; END WELD GEOMETRIA;%{PE}%R 4.1.16,%MKUKATPBASIS,%CCOMMENT,%VNORMAL,%P 2:END WELD GEOMETRIA
;ENDFOLD
;FOLD OUT 839 'R4 Soldando'  State= TRUE CONT;%{PE}%R 4.1.16,%MKUKATPBASIS,%COUT,%VOUTX,%P 2:839, 3:'R4 Soldando', 5:TRUE, 6:CONTINUE
CONTINUE
$OUT[839]=TRUE
;ENDFOLD
;FOLD PULSE 840 'R4 solda geometri concluida'  State= TRUE   Time= 2 sec;%{PE}%R 4.1.16,%MKUKATPBASIS,%COUT,%VPULSE,%P 2:840, 3:'R4 solda geometri concluida', 5:TRUE, 6:, 8:2
PULSE($OUT[840], TRUE,2)
;ENDFOLD

;FOLD PTP p1305 CONT Vel= 100 % PDAT130 Tool[1]:GUN C1 Base[2]:Accelo;%{PE}%R 4.1.16,%MKUKATPBASIS,%CMOVE,%VPTP,%P 1:PTP, 2:p1305, 3:C_PTP, 5:100, 7:PDAT130
$BWDSTART = FALSE
PDAT_ACT=PPDAT130
BAS(#PTP_DAT)
FDAT_ACT=Fp1305
BAS(#FRAMES)
BAS(#VEL_PTP,100)
PTP Xp1305 C_PTP
;ENDFOLD
;FOLD PTP p1307 CONT Vel= 100 % PDAT132 Tool[1]:GUN C1 Base[2]:Accelo;%{PE}%R 4.1.16,%MKUKATPBASIS,%CMOVE,%VPTP,%P 1:PTP, 2:p1307, 3:C_PTP, 5:100, 7:PDAT132
$BWDSTART = FALSE
PDAT_ACT=PPDAT132
BAS(#PTP_DAT)
FDAT_ACT=Fp1307
BAS(#FRAMES)
BAS(#VEL_PTP,100)
PTP Xp1307 C_PTP
;ENDFOLD

;FOLD PTP p1306  Vel= 100 % PDAT131 Tool[1]:GUN C1 Base[2]:Accelo;%{PE}%R 4.1.16,%MKUKATPBASIS,%CMOVE,%VPTP,%P 1:PTP, 2:p1306, 3:, 5:100, 7:PDAT131
$BWDSTART = FALSE
PDAT_ACT=PPDAT131
BAS(#PTP_DAT)
FDAT_ACT=Fp1306
BAS(#FRAMES)
BAS(#VEL_PTP,100)
PTP Xp1306
;ENDFOLD

;FOLD OUT 841 'Solic Lib. Soldar Respot Final'  State= TRUE ;%{PE}%R 4.1.16,%MKUKATPBASIS,%COUT,%VOUTX,%P 2:841, 3:'Solic Lib. Soldar Respot Final', 5:TRUE, 6:
$OUT[841]=TRUE
;ENDFOLD
;FOLD OUT 839 'R4 Soldando'  State= TRUE ;%{PE}%R 4.1.16,%MKUKATPBASIS,%COUT,%VOUTX,%P 2:839, 3:'R4 Soldando', 5:TRUE, 6:
$OUT[839]=TRUE
;ENDFOLD
;FOLD WAIT FOR IN 841 'Sinal de Anti-colisão para CLP'  State= TRUE ;%{PE}%R 4.1.16,%MKUKATPBASIS,%CWAIT_FOR,%VWAIT_FOR,%P 1:0, 2:841, 3:'Sinal de Anti-colisão para CLP', 5:TRUE, 6:
WAIT FOR $IN[841]==TRUE
;ENDFOLD
;FOLD OUT 839 'R4 Soldando'  State= FALSE ;%{PE}%R 4.1.16,%MKUKATPBASIS,%COUT,%VOUTX,%P 2:839, 3:'R4 Soldando', 5:FALSE, 6:
$OUT[839]=FALSE
;ENDFOLD
;FOLD OUT 841 'Solic Lib. Soldar Respot Final'  State= FALSE ;%{PE}%R 4.1.16,%MKUKATPBASIS,%COUT,%VOUTX,%P 2:841, 3:'Solic Lib. Soldar Respot Final', 5:FALSE, 6:
$OUT[841]=FALSE
;ENDFOLD
;FOLD OUT 840 'R4 solda geometri concluida'  State= FALSE ;%{PE}%R 4.1.16,%MKUKATPBASIS,%COUT,%VOUTX,%P 2:840, 3:'R4 solda geometri concluida', 5:FALSE, 6:
$OUT[840]=FALSE
;ENDFOLD
;FOLD OUT 848 'Area de Solda'  State= FALSE CONT;%{PE}%R 4.1.16,%MKUKATPBASIS,%COUT,%VOUTX,%P 2:848, 3:'Area de Solda', 5:FALSE, 6:CONTINUE
CONTINUE
$OUT[848]=FALSE
;ENDFOLD

;FOLD PULSE 844 'R4 solda RESPOT concluida'  State= TRUE   Time= 3 sec;%{PE}%R 4.1.16,%MKUKATPBASIS,%COUT,%VPULSE,%P 2:844, 3:'R4 solda RESPOT concluida', 5:TRUE, 6:, 8:3
PULSE($OUT[844], TRUE,3)
;ENDFOLD

;FOLD OUT 848 'Area de Solda'  State= TRUE ;%{PE}%R 4.1.16,%MKUKATPBASIS,%COUT,%VOUTX,%P 2:848, 3:'Area de Solda', 5:TRUE, 6:
$OUT[848]=TRUE
;ENDFOLD

END

--- ps_604c1.dat ---
&ACCESS RVO2
&REL 166
&COMMENT Geom C1 Accelo Atual sem o PTO 60-0682
DEFDAT  PS_604C1
;FOLD EXTERNAL DECLARATIONS;%{PE}%V2.2.2,%MKUKATPBASIS,%CEXT,%VCOMMON,%P
;FOLD BAS EXT;%{PE}%V2.2.2,%MKUKATPBASIS,%CEXT,%VEXT,%P
EXT  BAS (BAS_COMMAND  :IN,REAL  :IN )
DECL INT SUCCESS
;ENDFOLD
;FOLD A10 EXT;%{E}%V2.2.2,%MKUKATPARC,%CEXT,%VEXT,%P
EXT  A10 (A_CMD_T  :IN,A_STRT_T  :IN,A_WELD_T  :IN,A_END_T  :IN,INT  :IN )
;ENDFOLD
;FOLD A20 EXT;%{E}%V2.2.2,%MKUKATPA20,%CEXT,%VEXT,%P
EXT  A20 (INT  :IN,WELD_ST  :IN,WELD_FI  :IN,INT  :IN )
;ENDFOLD
;FOLD GRIPPER EXT;%{E}%V2.2.2,%MKUKATPGRIPPER,%CEXT,%VEXT,%P
EXT  H50 (INT  :IN,INT  :IN,INT  :IN,GRP_TYP  :IN )
;ENDFOLD
;FOLD SPOT EXT;%{E}%V2.2.2,%MKUKATPSPOT,%CEXT,%VEXT,%P
EXT  USERSPOT (S_COMMAND  :IN,SPOT_TYPE  :IN )
;ENDFOLD
;FOLD TOUCHSENSE EXT;%{E}%V2.2.2,%MKUKATPTS,%CEXT,%VEXT,%P
EXT  H70 (INT  :IN,SRCH_TYP_2  :OUT,E6POS  :IN,SRCH_TYP_3  :IN,SRCH_TYP_2  :IN,SRCH_TYP_2  :IN,SRCH_TYP_2  :IN,SRCH_TYP_2  :IN,SRCH_TYP_2  :IN,INT  :IN )
;ENDFOLD
;FOLD USER EXT;%{}%V2.2.2,%MKUKATPUSER,%CEXT,%VEXT,%P
;Make here your modifications
;ENDFOLD
;ENDFOLD

;# ============ START PATH : swp_p13060r4_ltc_geo_c1 =============
DECL BASIS_SUGG_T LAST_BASIS={POINT1[] "p1308                   ",POINT2[] "p1308                   ",CP_PARAMS[] "CPDAT0                  ",PTP_PARAMS[] "PDAT133                 ",CONT[] "C_PTP                   ",CP_VEL[] "2.0                     ",PTP_VEL[] "80                      "}
DECL E6POS Xp1325={x -664.33252,y 791.078308,z 1371.44495,a 63.5197105,b 34.798481,c -89.5357285,s 2,t 42,e1 0.0,e2 0.0,e3 0.0,e4 0.0,e5 0.0,e6 0.0}
DECL FDAT Fp1325={TOOL_NO 1,BASE_NO 2,IPO_FRAME #BASE}
DECL PDAT PPDAT36={VEL 100.0,ACC 80.0,APO_DIST 100.0}
DECL E6POS Xp1326={x 509.065491,y 788.343628,z 1125.00305,a 78.9254227,b -26.6650105,c -65.7811127,s 2,t 43,e1 0.0,e2 0.0,e3 0.0,e4 0.0,e5 0.0,e6 0.0}
DECL FDAT Fp1326={TOOL_NO 1,BASE_NO 2,IPO_FRAME #BASE}
DECL PDAT PPDAT37={VEL 100.0,ACC 80.0,APO_DIST 100.0}
DECL E6POS Xswp_60_0806={x 511.212494,y 873.906311,z 1145.47803,a 73.4269638,b -0.701606572,c -67.3485565,s 2,t 43,e1 0.0,e2 0.0,e3 0.0,e4 0.0,e5 0.0,e6 0.0}
DECL FDAT Fswp_60_0806={TOOL_NO 1,BASE_NO 2,IPO_FRAME #BASE}
DECL PDAT PPDAT38={VEL 100.0,ACC 100.0,APO_DIST 100.0}
DECL E6POS Xswp_60_0804={x 497.138,y 881.864929,z 1121.92603,a 73.5548782,b -0.462380588,c -68.111763,s 2,t 43,e1 0.0,e2 0.0,e3 0.0,e4 0.0,e5 0.0,e6 0.0}
DECL FDAT Fswp_60_0804={TOOL_NO 1,BASE_NO 2,IPO_FRAME #BASE}
DECL PDAT PPDAT39={VEL 100.0,ACC 100.0,APO_DIST 100.0}
DECL E6POS Xp1317={x 490.735687,y 860.807312,z 1094.17395,a 68.8672638,b -13.4404297,c -66.8604965,s 2,t 43,e1 0.0,e2 0.0,e3 0.0,e4 0.0,e5 0.0,e6 0.0}
DECL FDAT Fp1317={TOOL_NO 1,BASE_NO 2,IPO_FRAME #BASE}
DECL PDAT PPDAT40={VEL 100.0,ACC 80.0,APO_DIST 2.0}
DECL E6POS Xswp_60_0802={x 474.677002,y 887.624878,z 1077.37598,a 72.1530533,b -3.70327711,c -63.4271393,s 2,t 43,e1 0.0,e2 0.0,e3 0.0,e4 0.0,e5 0.0,e6 0.0}
DECL FDAT Fswp_60_0802={TOOL_NO 1,BASE_NO 2,IPO_FRAME #BASE}
DECL PDAT PPDAT41={VEL 100.0,ACC 100.0,APO_DIST 100.0}
DECL E6POS Xswp_60_0798={x 427.168915,y 899.093811,z 997.465515,a 65.9514389,b -11.1565504,c -63.5836182,s 2,t 43,e1 0.0,e2 0.0,e3 0.0,e4 0.0,e5 0.0,e6 0.0}
DECL FDAT Fswp_60_0798={TOOL_NO 1,BASE_NO 2,IPO_FRAME #BASE}
DECL PDAT PPDAT43={VEL 100.0,ACC 100.0,APO_DIST 100.0}
DECL E6POS Xswp_60_0794={x 403.701813,y 901.828125,z 948.634827,a 66.5146637,b -7.58480978,c -61.9485512,s 2,t 43,e1 0.0,e2 0.0,e3 0.0,e4 0.0,e5 0.0,e6 0.0}
DECL FDAT Fswp_60_0794={TOOL_NO 1,BASE_NO 2,IPO_FRAME #BASE}
DECL PDAT PPDAT44={VEL 100.0,ACC 100.0,APO_DIST 100.0}
DECL E6POS Xp1282={x 421.36319,y 868.844116,z 954.054626,a 67.8700027,b -12.8819599,c -61.6052208,s 2,t 43,e1 0.0,e2 0.0,e3 0.0,e4 0.0,e5 0.0,e6 0.0}
DECL FDAT Fp1282={TOOL_NO 1,BASE_NO 2,IPO_FRAME #BASE}
DECL PDAT PP_OLP77={VEL 100.0,ACC 80.0,APO_DIST 10.0}
DECL E6POS Xp1316={x 383.631592,y 874.919617,z 889.793579,a 72.5711288,b -6.59166288,c -62.5001907,s 2,t 43,e1 0.0,e2 0.0,e3 0.0,e4 0.0,e5 0.0,e6 0.0}
DECL FDAT Fp1316={TOOL_NO 1,BASE_NO 2,IPO_FRAME #BASE}
DECL PDAT PPDAT45={VEL 100.0,ACC 80.0,APO_DIST 10.0}
DECL E6POS Xswp_60_0792={x 373.974609,y 909.131592,z 893.5896,a 69.6701508,b -3.07000494,c -62.354351,s 2,t 43,e1 0.0,e2 0.0,e3 0.0,e4 0.0,e5 0.0,e6 0.0}
DECL FDAT Fswp_60_0792={TOOL_NO 1,BASE_NO 2,IPO_FRAME #BASE}
DECL PDAT PPDAT46={VEL 100.0,ACC 100.0,APO_DIST 100.0}
DECL E6POS Xswp_60_0790={x 352.678314,y 911.065979,z 854.552795,a 69.4925232,b -1.88326502,c -62.7122803,s 2,t 43,e1 0.0,e2 0.0,e3 0.0,e4 0.0,e5 0.0,e6 0.0}
DECL FDAT Fswp_60_0790={TOOL_NO 1,BASE_NO 2,IPO_FRAME #BASE}
DECL PDAT PPDAT47={VEL 100.0,ACC 100.0,APO_DIST 100.0}
DECL E6POS Xswp_60_0788={x 339.479706,y 912.431519,z 828.406494,a 74.7219772,b 2.6001091,c -62.7704887,s 2,t 43,e1 0.0,e2 0.0,e3 0.0,e4 0.0,e5 0.0,e6 0.0}
DECL FDAT Fswp_60_0788={TOOL_NO 1,BASE_NO 2,IPO_FRAME #BASE}
DECL PDAT PPDAT48={VEL 100.0,ACC 100.0,APO_DIST 100.0}
DECL E6POS Xp1321={x 341.286713,y 882.1474,z 817.836121,a 70.0848618,b -11.91047,c -62.0434914,s 2,t 43,e1 0.0,e2 0.0,e3 0.0,e4 0.0,e5 0.0,e6 0.0}
DECL FDAT Fp1321={TOOL_NO 1,BASE_NO 2,IPO_FRAME #BASE}
DECL PDAT PPDAT49={VEL 100.0,ACC 80.0,APO_DIST 100.0}
DECL E6POS Xswp_60_0786={x 315.640503,y 916.632202,z 780.782104,a 73.0588074,b -1.074435,c -63.3973083,s 2,t 43,e1 0.0,e2 0.0,e3 0.0,e4 0.0,e5 0.0,e6 0.0}
DECL FDAT Fswp_60_0786={TOOL_NO 1,BASE_NO 2,IPO_FRAME #BASE}
DECL PDAT PPDAT50={VEL 100.0,ACC 100.0,APO_DIST 100.0}
DECL E6POS Xp1322={x 308.105713,y 873.905273,z 742.801514,a 70.0945435,b -11.8402796,c -61.8813286,s 2,t 43,e1 0.0,e2 0.0,e3 0.0,e4 0.0,e5 0.0,e6 0.0}
DECL FDAT Fp1322={TOOL_NO 1,BASE_NO 2,IPO_FRAME #BASE}
DECL PDAT PPDAT51={VEL 100.0,ACC 80.0,APO_DIST 100.0}
DECL E6POS Xp1323={x 289.292786,y 904.557983,z 722.148315,a 70.97966,b -3.04607892,c -62.6529007,s 2,t 43,e1 0.0,e2 0.0,e3 0.0,e4 0.0,e5 0.0,e6 0.0}
DECL FDAT Fp1323={TOOL_NO 1,BASE_NO 2,IPO_FRAME #BASE}
DECL PDAT PPDAT52={VEL 100.0,ACC 80.0,APO_DIST 100.0}
DECL E6POS Xswp_60_0782={x 286.730103,y 933.546814,z 710.258484,a 72.1367035,b 4.24815083,c -61.9066811,s 2,t 43,e1 0.0,e2 0.0,e3 0.0,e4 0.0,e5 0.0,e6 0.0}
DECL FDAT Fswp_60_0782={TOOL_NO 1,BASE_NO 2,IPO_FRAME #BASE}
DECL PDAT PPDAT53={VEL 100.0,ACC 100.0,APO_DIST 100.0}
DECL E6POS Xp1327={x 286.896912,y 901.282471,z 721.870728,a 66.3050079,b -11.9102802,c -62.0441093,s 2,t 43,e1 0.0,e2 0.0,e3 0.0,e4 0.0,e5 0.0,e6 0.0}
DECL FDAT Fp1327={TOOL_NO 1,BASE_NO 2,IPO_FRAME #BASE}
DECL PDAT PPDAT55={VEL 100.0,ACC 80.0,APO_DIST 100.0}
DECL E6POS Xp1328={x 206.840805,y 882.34137,z 764.955627,a 66.3052673,b -11.9082699,c -62.0422592,s 2,t 43,e1 0.0,e2 0.0,e3 0.0,e4 0.0,e5 0.0,e6 0.0}
DECL FDAT Fp1328={TOOL_NO 1,BASE_NO 2,IPO_FRAME #BASE}
DECL PDAT PPDAT56={VEL 100.0,ACC 80.0,APO_DIST 100.0}
DECL E6POS Xp1310={x 164.661804,y 887.389221,z 681.890686,a 66.3055801,b -11.9089699,c -62.0430717,s 2,t 43,e1 0.0,e2 0.0,e3 0.0,e4 0.0,e5 0.0,e6 0.0}
DECL FDAT Fp1310={TOOL_NO 1,BASE_NO 2,IPO_FRAME #BASE}
DECL PDAT PP_OLP78={VEL 100.0,ACC 80.0,APO_DIST 10.0}
DECL E6POS XP1226={x 493.117493,y 845.016479,z 1088.927,a 67.585083,b -12.6274004,c -65.7208862,s 2,t 43,e1 0.0,e2 0.0,e3 0.0,e4 0.0,e5 0.0,e6 0.0}
DECL FDAT Fp1226={TOOL_NO 1,BASE_NO 2,IPO_FRAME #BASE}
DECL PDAT PPDAT57={VEL 100.0,ACC 80.0,APO_DIST 10.0}
DECL E6POS XP1227={x 411.549896,y 859.407288,z 1119.46997,a 67.5851822,b -12.62745,c -65.7212067,s 2,t 43,e1 0.0,e2 0.0,e3 0.0,e4 0.0,e5 0.0,e6 0.0}
DECL FDAT Fp1227={TOOL_NO 1,BASE_NO 2,IPO_FRAME #BASE}
DECL PDAT PPDAT58={VEL 100.0,ACC 80.0,APO_DIST 10.0}
DECL E6POS XP1228={x 346.094513,y 858.244324,z 1036.22302,a 67.5846024,b -12.62815,c -65.7201996,s 2,t 43,e1 0.0,e2 0.0,e3 0.0,e4 0.0,e5 0.0,e6 0.0}
DECL FDAT Fp1228={TOOL_NO 1,BASE_NO 2,IPO_FRAME #BASE}
DECL PDAT PPDAT59={VEL 100.0,ACC 80.0,APO_DIST 10.0}
DECL E6POS XP1229={x 437.514099,y 862.001526,z 1006.414,a 67.5844574,b -12.6285801,c -65.7204132,s 2,t 43,e1 0.0,e2 0.0,e3 0.0,e4 0.0,e5 0.0,e6 0.0}
DECL FDAT Fp1229={TOOL_NO 1,BASE_NO 2,IPO_FRAME #BASE}
DECL PDAT PPDAT60={VEL 100.0,ACC 80.0,APO_DIST 10.0}
DECL E6POS XP1230={x 418.648499,y 903.963379,z 978.689514,a 56.6214104,b -27.0063992,c -58.1820488,s 2,t 43,e1 0.0,e2 0.0,e3 0.0,e4 0.0,e5 0.0,e6 0.0}
DECL FDAT Fp1230={TOOL_NO 1,BASE_NO 2,IPO_FRAME #BASE}
DECL PDAT PPDAT61={VEL 100.0,ACC 100.0,APO_DIST 100.0}
DECL E6POS XP1231={x 240.077194,y 877.396423,z 627.976318,a 66.3055115,b -11.9088202,c -62.0430908,s 2,t 43,e1 0.0,e2 0.0,e3 0.0,e4 0.0,e5 0.0,e6 0.0}
DECL FDAT Fp1231={TOOL_NO 1,BASE_NO 2,IPO_FRAME #BASE}
DECL PDAT PPDAT62={VEL 100.0,ACC 80.0,APO_DIST 10.0}
DECL E6POS Xswp_60_0779={x 245.274307,y 923.200684,z 627.302979,a 70.4701538,b -3.91291094,c -62.6390686,s 2,t 43,e1 0.0,e2 0.0,e3 0.0,e4 0.0,e5 0.0,e6 0.0}
DECL FDAT Fswp_60_0779={TOOL_NO 1,BASE_NO 2,IPO_FRAME #BASE}
DECL PDAT PPDAT63={VEL 100.0,ACC 100.0,APO_DIST 100.0}
DECL E6POS Xswp_60_0777={x 228.413193,y 924.177979,z 591.891785,a 70.9297867,b -3.02607894,c -62.6661911,s 2,t 43,e1 0.0,e2 0.0,e3 0.0,e4 0.0,e5 0.0,e6 0.0}
DECL FDAT Fswp_60_0777={TOOL_NO 1,BASE_NO 2,IPO_FRAME #BASE}
DECL PDAT PPDAT64={VEL 100.0,ACC 100.0,APO_DIST 100.0}
DECL E6POS Xswp_60_0775={x 215.485504,y 921.907715,z 562.566406,a 71.8485413,b -1.24762106,c -62.700161,s 2,t 43,e1 0.0,e2 0.0,e3 0.0,e4 0.0,e5 0.0,e6 0.0}
DECL FDAT Fswp_60_0775={TOOL_NO 1,BASE_NO 2,IPO_FRAME #BASE}
DECL PDAT PPDAT65={VEL 100.0,ACC 100.0,APO_DIST 100.0}
DECL E6POS XSWP_60_0773={x 208.627396,y 917.088928,z 530.926392,a 100.930603,b 39.4170418,c -52.80616,s 2,t 43,e1 0.0,e2 0.0,e3 0.0,e4 0.0,e5 0.0,e6 0.0}
DECL FDAT FSWP_60_0773={TOOL_NO 1,BASE_NO 2,IPO_FRAME #BASE}
DECL PDAT PPDAT66={VEL 100.0,ACC 100.0,APO_DIST 100.0}
DECL E6POS Xp1232={x 221.027603,y 886.39093,z 553.484314,a 105.373901,b 36.6275291,c -50.0648804,s 2,t 43,e1 0.0,e2 0.0,e3 0.0,e4 0.0,e5 0.0,e6 0.0}
DECL FDAT Fp1232={TOOL_NO 1,BASE_NO 2,IPO_FRAME #BASE}
DECL PDAT PP_OLP79={VEL 100.0,ACC 85.0,APO_DIST 10.0}
DECL E6POS XSWP_60_0199={x 189.641098,y 883.742493,z 523.760193,a 178.942703,b 65.2382965,c 15.5449896,s 2,t 11,e1 0.0,e2 0.0,e3 0.0,e4 0.0,e5 0.0,e6 0.0}
DECL FDAT FSWP_60_0199={TOOL_NO 1,BASE_NO 2,IPO_FRAME #BASE}
DECL PDAT PPDAT67={VEL 100.0,ACC 100.0,APO_DIST 100.0}
DECL E6POS Xswp_60_0193={x 139.549896,y 698.185425,z 528.21283,a 165.181503,b 69.6868362,c -11.9993401,s 2,t 11,e1 0.0,e2 0.0,e3 0.0,e4 0.0,e5 0.0,e6 0.0}
DECL FDAT Fswp_60_0193={TOOL_NO 1,BASE_NO 2,IPO_FRAME #BASE}
DECL PDAT PPDAT68={VEL 100.0,ACC 100.0,APO_DIST 100.0}
DECL E6POS XSWP_60_0185={x 118.644699,y 516.663879,z 526.738403,a 179.998596,b 62.8476486,c 4.22270298,s 2,t 11,e1 0.0,e2 0.0,e3 0.0,e4 0.0,e5 0.0,e6 0.0}
DECL FDAT FSWP_60_0185={TOOL_NO 1,BASE_NO 2,IPO_FRAME #BASE}
DECL PDAT PPDAT69={VEL 100.0,ACC 100.0,APO_DIST 100.0}
DECL E6POS Xswp_60_0167={x 97.5838776,y 90.6914063,z 531.459778,a 179.996094,b 62.9335403,c 3.64204693,s 2,t 11,e1 0.0,e2 0.0,e3 0.0,e4 0.0,e5 0.0,e6 0.0}
DECL FDAT Fswp_60_0167={TOOL_NO 1,BASE_NO 2,IPO_FRAME #BASE}
DECL PDAT PPDAT70={VEL 100.0,ACC 100.0,APO_DIST 100.0}
DECL E6POS XSWP_60_0103={x 33.1900482,y 251.159698,z 159.220795,a 62.1840096,b -81.8501129,c -69.2860031,s 2,t 43,e1 0.0,e2 0.0,e3 0.0,e4 0.0,e5 0.0,e6 0.0}
DECL FDAT FSWP_60_0103={TOOL_NO 1,BASE_NO 2,IPO_FRAME #BASE}
DECL PDAT PPDAT71={VEL 100.0,ACC 100.0,APO_DIST 100.0}
DECL E6POS XSWP_60_0115={x 44.7215118,y 454.82019,z 144.828903,a 79.1381836,b -54.5401001,c -83.5403366,s 2,t 43,e1 0.0,e2 0.0,e3 0.0,e4 0.0,e5 0.0,e6 0.0}
DECL FDAT FSWP_60_0115={TOOL_NO 1,BASE_NO 2,IPO_FRAME #BASE}
DECL PDAT PPDAT72={VEL 100.0,ACC 100.0,APO_DIST 100.0}
DECL E6POS XSWP_60_0117={x 57.0946198,y 676.087585,z 155.435699,a -91.4680405,b -65.216568,c 82.8926086,s 2,t 43,e1 0.0,e2 0.0,e3 0.0,e4 0.0,e5 0.0,e6 0.0}
DECL FDAT FSWP_60_0117={TOOL_NO 1,BASE_NO 2,IPO_FRAME #BASE}
DECL PDAT PPDAT73={VEL 100.0,ACC 100.0,APO_DIST 100.0}
DECL E6POS Xswp_60_0119={x 59.2961311,y 701.344788,z 166.678207,a 37.52174,b -85.3697815,c -43.2334595,s 2,t 43,e1 0.0,e2 0.0,e3 0.0,e4 0.0,e5 0.0,e6 0.0}
DECL FDAT Fswp_60_0119={TOOL_NO 1,BASE_NO 2,IPO_FRAME #BASE}
DECL PDAT PPDAT74={VEL 100.0,ACC 100.0,APO_DIST 100.0}
DECL E6POS Xswp_60_0121={x 64.723671,y 737.429871,z 176.719803,a 1.01746702,b -86.1406174,c -6.63438082,s 2,t 43,e1 0.0,e2 0.0,e3 0.0,e4 0.0,e5 0.0,e6 0.0}
DECL FDAT Fswp_60_0121={TOOL_NO 1,BASE_NO 2,IPO_FRAME #BASE}
DECL PDAT PPDAT75={VEL 100.0,ACC 100.0,APO_DIST 100.0}
DECL E6POS Xswp_60_0123={x 70.7058487,y 770.983276,z 185.503601,a 37.5734406,b -85.3683929,c -43.2851906,s 2,t 43,e1 0.0,e2 0.0,e3 0.0,e4 0.0,e5 0.0,e6 0.0}
DECL FDAT Fswp_60_0123={TOOL_NO 1,BASE_NO 2,IPO_FRAME #BASE}
DECL PDAT PPDAT76={VEL 100.0,ACC 100.0,APO_DIST 100.0}
DECL E6POS XSWP_60_0127={x 85.5572662,y 829.834106,z 198.907898,a 0.0115195401,b -84.8815536,c -10.1871996,s 2,t 43,e1 0.0,e2 0.0,e3 0.0,e4 0.0,e5 0.0,e6 0.0}
DECL FDAT FSWP_60_0127={TOOL_NO 1,BASE_NO 2,IPO_FRAME #BASE}
DECL PDAT PPDAT77={VEL 100.0,ACC 100.0,APO_DIST 100.0}
DECL E6POS XP1233={x 196.427902,y 797.649475,z 561.333618,a 178.940201,b 65.2386322,c 15.5427704,s 2,t 11,e1 0.0,e2 0.0,e3 0.0,e4 0.0,e5 0.0,e6 0.0}
DECL FDAT Fp1233={TOOL_NO 1,BASE_NO 2,IPO_FRAME #BASE}
DECL PDAT PPDAT78={VEL 100.0,ACC 85.0,APO_DIST 10.0}
DECL E6POS XP1234={x 194.426697,y 709.277771,z 585.929626,a 175.884293,b 65.1324463,c 2.56119204,s 2,t 11,e1 0.0,e2 0.0,e3 0.0,e4 0.0,e5 0.0,e6 0.0}
DECL FDAT Fp1234={TOOL_NO 1,BASE_NO 2,IPO_FRAME #BASE}
DECL PDAT PPDAT79={VEL 100.0,ACC 85.0,APO_DIST 10.0}
DECL E6POS XP1235={x 143.495499,y 592.479614,z 531.168823,a 175.481201,b 65.6446304,c -1.18967199,s 2,t 11,e1 0.0,e2 0.0,e3 0.0,e4 0.0,e5 0.0,e6 0.0}
DECL FDAT Fp1235={TOOL_NO 1,BASE_NO 2,IPO_FRAME #BASE}
DECL PDAT PPDAT80={VEL 100.0,ACC 85.0,APO_DIST 10.0}
DECL E6POS XP1236={x 156.862396,y 516.407227,z 580.971191,a 179.998306,b 62.8476715,c 4.22266483,s 2,t 11,e1 0.0,e2 0.0,e3 0.0,e4 0.0,e5 0.0,e6 0.0}
DECL FDAT Fp1236={TOOL_NO 1,BASE_NO 2,IPO_FRAME #BASE}
DECL PDAT PPDAT81={VEL 100.0,ACC 85.0,APO_DIST 10.0}
DECL E6POS XP1237={x 254.760406,y 501.1203,z 792.022827,a 173.335602,b 72.0107269,c -1.42356503,s 2,t 11,e1 0.0,e2 0.0,e3 0.0,e4 0.0,e5 0.0,e6 0.0}
DECL FDAT Fp1237={TOOL_NO 1,BASE_NO 2,IPO_FRAME #BASE}
DECL PDAT PPDAT82={VEL 100.0,ACC 85.0,APO_DIST 20.0}
DECL E6POS XP1238={x 257.313507,y 243.034302,z 797.192383,a 173.344406,b 72.0115509,c -1.41443896,s 2,t 11,e1 0.0,e2 0.0,e3 0.0,e4 0.0,e5 0.0,e6 0.0}
DECL FDAT Fp1238={TOOL_NO 1,BASE_NO 2,IPO_FRAME #BASE}
DECL PDAT PPDAT83={VEL 100.0,ACC 85.0,APO_DIST 20.0}
DECL E6POS XP1239={x 144.798004,y 123.605598,z 592.043274,a 179.228195,b 65.0072174,c 3.1434319,s 2,t 11,e1 0.0,e2 0.0,e3 0.0,e4 0.0,e5 0.0,e6 0.0}
DECL FDAT Fp1239={TOOL_NO 1,BASE_NO 2,IPO_FRAME #BASE}
DECL PDAT PPDAT84={VEL 100.0,ACC 85.0,APO_DIST 10.0}
DECL E6POS XP1240={x 179.080597,y 132.7565,z 671.88739,a 178.561401,b 69.1954422,c 0.682946622,s 2,t 11,e1 0.0,e2 0.0,e3 0.0,e4 0.0,e5 0.0,e6 0.0}
DECL FDAT Fp1240={TOOL_NO 1,BASE_NO 2,IPO_FRAME #BASE}
DECL PDAT PPDAT85={VEL 100.0,ACC 85.0,APO_DIST 10.0}
DECL E6POS XP1241={x -440.210693,y 288.873108,z 705.667175,a 145.069901,b 65.5228577,c -22.6158199,s 2,t 10,e1 0.0,e2 0.0,e3 0.0,e4 0.0,e5 0.0,e6 0.0}
DECL FDAT Fp1241={TOOL_NO 1,BASE_NO 2,IPO_FRAME #BASE}
DECL PDAT PPDAT86={VEL 100.0,ACC 85.0,APO_DIST 20.0}
DECL E6POS XP1242={x -392.090698,y 312.830902,z 86.7444916,a -51.7184601,b -78.2493668,c 42.6988411,s 2,t 42,e1 0.0,e2 0.0,e3 0.0,e4 0.0,e5 0.0,e6 0.0}
DECL FDAT Fp1242={TOOL_NO 1,BASE_NO 2,IPO_FRAME #BASE}
DECL PDAT PPDAT87={VEL 100.0,ACC 85.0,APO_DIST 20.0}
DECL E6POS XP1243={x 41.6715813,y 247.586899,z 121.7099,a 47.1596909,b -83.5169983,c -54.4612617,s 2,t 43,e1 0.0,e2 0.0,e3 0.0,e4 0.0,e5 0.0,e6 0.0}
DECL FDAT Fp1243={TOOL_NO 1,BASE_NO 2,IPO_FRAME #BASE}
DECL PDAT PPDAT88={VEL 100.0,ACC 85.0,APO_DIST 10.0}
DECL E6POS XP1244={x 43.6024094,y 388.292389,z 103.355003,a 47.1433296,b -83.5185623,c -54.4453392,s 2,t 43,e1 0.0,e2 0.0,e3 0.0,e4 0.0,e5 0.0,e6 0.0}
DECL FDAT Fp1244={TOOL_NO 1,BASE_NO 2,IPO_FRAME #BASE}
DECL PDAT PPDAT89={VEL 100.0,ACC 85.0,APO_DIST 10.0}
DECL E6POS XP1245={x 40.8675194,y 246.726395,z 111.085098,a 47.1441689,b -83.5185089,c -54.4452019,s 2,t 43,e1 0.0,e2 0.0,e3 0.0,e4 0.0,e5 0.0,e6 0.0}
DECL FDAT Fp1245={TOOL_NO 1,BASE_NO 2,IPO_FRAME #BASE}
DECL PDAT PPDAT90={VEL 100.0,ACC 85.0,APO_DIST 10.0}
DECL E6POS XP1246={x 43.6024094,y 388.292389,z 103.355003,a 47.1433296,b -83.5185623,c -54.4453392,s 2,t 43,e1 0.0,e2 0.0,e3 0.0,e4 0.0,e5 0.0,e6 0.0}
DECL FDAT Fp1246={TOOL_NO 1,BASE_NO 2,IPO_FRAME #BASE}
DECL PDAT PPDAT91={VEL 100.0,ACC 85.0,APO_DIST 10.0}
DECL E6POS XP1247={x -387.1185,y 444.809814,z 131.930099,a 47.1437798,b -83.5184402,c -54.4458389,s 2,t 42,e1 0.0,e2 0.0,e3 0.0,e4 0.0,e5 0.0,e6 0.0}
DECL FDAT Fp1247={TOOL_NO 1,BASE_NO 2,IPO_FRAME #BASE}
DECL PDAT PPDAT92={VEL 100.0,ACC 85.0,APO_DIST 20.0}
DECL E6POS XP1248={x -352.059601,y 725.168518,z 105.862503,a 47.1415901,b -83.518158,c -54.4438095,s 2,t 42,e1 0.0,e2 0.0,e3 0.0,e4 0.0,e5 0.0,e6 0.0}
DECL FDAT Fp1248={TOOL_NO 1,BASE_NO 2,IPO_FRAME #BASE}
DECL PDAT PPDAT93={VEL 100.0,ACC 85.0,APO_DIST 20.0}
DECL E6POS XP1249={x 65.9035492,y 679.190002,z 102.245201,a -88.8125305,b -70.7309723,c 80.429657,s 2,t 43,e1 0.0,e2 0.0,e3 0.0,e4 0.0,e5 0.0,e6 0.0}
DECL FDAT Fp1249={TOOL_NO 1,BASE_NO 2,IPO_FRAME #BASE}
DECL PDAT PPDAT94={VEL 100.0,ACC 85.0,APO_DIST 10.0}
DECL E6POS Xswp_60_0125={x 78.2941132,y 801.625,z 193.599197,a 37.549511,b -85.3698578,c -43.2609711,s 2,t 43,e1 0.0,e2 0.0,e3 0.0,e4 0.0,e5 0.0,e6 0.0}
DECL FDAT Fswp_60_0125={TOOL_NO 1,BASE_NO 2,IPO_FRAME #BASE}
DECL PDAT PPDAT95={VEL 100.0,ACC 100.0,APO_DIST 100.0}
DECL E6POS XP1250={x 91.2592163,y 811.730286,z 137.247101,a -3.35188389,b -82.4603882,c -7.55397987,s 2,t 43,e1 0.0,e2 0.0,e3 0.0,e4 0.0,e5 0.0,e6 0.0}
DECL FDAT Fp1250={TOOL_NO 1,BASE_NO 2,IPO_FRAME #BASE}
DECL PDAT PPDAT96={VEL 100.0,ACC 85.0,APO_DIST 10.0}
DECL E6POS XP1251={x -323.091797,y 892.059387,z 192.601501,a -3.35227489,b -82.4598312,c -7.55339193,s 2,t 42,e1 0.0,e2 0.0,e3 0.0,e4 0.0,e5 0.0,e6 0.0}
DECL FDAT Fp1251={TOOL_NO 1,BASE_NO 2,IPO_FRAME #BASE}
DECL PDAT PPDAT97={VEL 100.0,ACC 85.0,APO_DIST 10.0}
DECL E6POS XP1252={x -715.440613,y 852.356384,z 113.869698,a 28.8778992,b -70.7833023,c -37.8725014,s 2,t 42,e1 0.0,e2 0.0,e3 0.0,e4 0.0,e5 0.0,e6 0.0}
DECL FDAT Fp1252={TOOL_NO 1,BASE_NO 2,IPO_FRAME #BASE}
DECL PDAT PPDAT98={VEL 100.0,ACC 85.0,APO_DIST 10.0}
DECL E6POS XP1275={x -718.189819,y 623.507874,z 1276.36694,a 67.2133636,b -4.25199986,c -101.8592,s 2,t 42,e1 0.0,e2 0.0,e3 0.0,e4 0.0,e5 0.0,e6 0.0}
DECL FDAT Fp1275={TOOL_NO 1,BASE_NO 2,IPO_FRAME #BASE}
DECL PDAT PPDAT104={VEL 100.0,ACC 80.0,APO_DIST 100.0}
DECL E6POS XP1286={x 207.319901,y 887.483826,z 556.34729,a 176.678497,b 66.9554672,c 13.1319199,s 2,t 11,e1 0.0,e2 0.0,e3 0.0,e4 0.0,e5 0.0,e6 0.0}
DECL FDAT Fp1286={TOOL_NO 1,BASE_NO 2,IPO_FRAME #BASE}
DECL PDAT PPDAT116={VEL 100.0,ACC 80.0,APO_DIST 100.0}
DECL E6POS XSWP_60_0785={x 298.163208,y 918.408081,z 743.191528,a 73.4181976,b 8.52011967,c -63.5458717,s 2,t 43,e1 0.0,e2 0.0,e3 0.0,e4 0.0,e5 0.0,e6 0.0}
DECL FDAT FSWP_60_0785={TOOL_NO 1,BASE_NO 2,IPO_FRAME #BASE}
DECL PDAT PPDAT117={VEL 100.0,ACC 100.0,APO_DIST 100.0}
DECL E6POS XP1287={x -1727.724,y 741.768616,z 413.36261,a 53.5088501,b 25.8493195,c -42.8503609,s 2,t 42,e1 0.0,e2 0.0,e3 0.0,e4 0.0,e5 0.0,e6 0.0}
DECL FDAT Fp1287={TOOL_NO 1,BASE_NO 2,IPO_FRAME #BASE}
DECL PDAT PPDAT118={VEL 100.0,ACC 80.0,APO_DIST 100.0}
DECL E6POS Xp1292={x 528.857422,y 819.397217,z 1132.078,a 79.3153763,b -25.89147,c -65.956337,s 2,t 43,e1 0.0,e2 0.0,e3 0.0,e4 0.0,e5 0.0,e6 0.0}
DECL FDAT Fp1292={TOOL_NO 1,BASE_NO 2,IPO_FRAME #BASE}
DECL PDAT PPDAT122={VEL 100.0,ACC 80.0,APO_DIST 100.0}
DECL E6POS Xp1293={x 486.596497,y 865.466675,z 1088.86804,a 73.0518112,b -19.1729794,c -63.9295502,s 2,t 43,e1 0.0,e2 0.0,e3 0.0,e4 0.0,e5 0.0,e6 0.0}
DECL FDAT Fp1293={TOOL_NO 1,BASE_NO 2,IPO_FRAME #BASE}
DECL PDAT PPDAT123={VEL 100.0,ACC 80.0,APO_DIST 100.0}
DECL E6POS Xswp_60_0803={x 452.408905,y 900.328918,z 1036.31494,a 69.1045532,b -12.6671,c -63.8056107,s 2,t 43,e1 0.0,e2 0.0,e3 0.0,e4 0.0,e5 0.0,e6 0.0}
DECL FDAT Fswp_60_0803={TOOL_NO 1,BASE_NO 2,IPO_FRAME #BASE}
DECL PDAT PPDAT124={VEL 100.0,ACC 100.0,APO_DIST 100.0}
DECL E6POS Xp1294={x 439.661407,y 839.448303,z 1022.94397,a 69.1042175,b -12.66675,c -63.8056297,s 2,t 43,e1 0.0,e2 0.0,e3 0.0,e4 0.0,e5 0.0,e6 0.0}
DECL FDAT Fp1294={TOOL_NO 1,BASE_NO 2,IPO_FRAME #BASE}
DECL PDAT PPDAT125={VEL 100.0,ACC 80.0,APO_DIST 100.0}
DECL E6POS Xp1295={x 275.033203,y 911.768372,z 680.668579,a 66.2555084,b -11.8890104,c -62.0573387,s 2,t 43,e1 0.0,e2 0.0,e3 0.0,e4 0.0,e5 0.0,e6 0.0}
DECL FDAT Fp1295={TOOL_NO 1,BASE_NO 2,IPO_FRAME #BASE}
DECL PDAT PPDAT126={VEL 100.0,ACC 80.0,APO_DIST 100.0}
DECL E6POS Xswp_60_0783={x 261.927307,y 927.338501,z 668.966919,a 66.255661,b -11.8886003,c -62.0566101,s 2,t 43,e1 0.0,e2 0.0,e3 0.0,e4 0.0,e5 0.0,e6 0.0}
DECL FDAT Fswp_60_0783={TOOL_NO 1,BASE_NO 2,IPO_FRAME #BASE}
DECL PDAT PPDAT127={VEL 100.0,ACC 100.0,APO_DIST 100.0}
DECL E6POS Xp1296={x 260.493011,y 878.723206,z 673.048523,a 66.2550812,b -11.8894901,c -62.0564995,s 2,t 43,e1 0.0,e2 0.0,e3 0.0,e4 0.0,e5 0.0,e6 0.0}
DECL FDAT Fp1296={TOOL_NO 1,BASE_NO 2,IPO_FRAME #BASE}
DECL PDAT PPDAT128={VEL 100.0,ACC 80.0,APO_DIST 100.0}
DECL E6POS Xp1304={x -194.8405,y 697.135925,z 794.950623,a 56.4149208,b -12.0441198,c -62.1975899,s 2,t 43,e1 0.0,e2 0.0,e3 0.0,e4 0.0,e5 0.0,e6 0.0}
DECL FDAT Fp1304={TOOL_NO 1,BASE_NO 2,IPO_FRAME #BASE}
DECL PDAT PPDAT129={VEL 100.0,ACC 80.0,APO_DIST 100.0}
DECL E6POS Xp1305={x -1167.27795,y 764.58728,z 44.8211708,a 13.4936304,b -44.326931,c -23.5247192,s 2,t 42,e1 0.0,e2 0.0,e3 0.0,e4 0.0,e5 0.0,e6 0.0}
DECL FDAT Fp1305={TOOL_NO 1,BASE_NO 2,IPO_FRAME #BASE}
DECL PDAT PPDAT130={VEL 100.0,ACC 80.0,APO_DIST 100.0}
DECL E6POS Xp1306={x -4006.80493,y 1991.11597,z 459.745514,a -84.1191406,b 2.5422709,c -49.1447296,s 2,t 34,e1 0.0,e2 0.0,e3 0.0,e4 0.0,e5 0.0,e6 0.0}
DECL FDAT Fp1306={TOOL_NO 1,BASE_NO 2,IPO_FRAME #BASE}
DECL PDAT PPDAT131={VEL 100.0,ACC 80.0,APO_DIST 100.0}
DECL E6POS XP1307={x -2114.36304,y 715.972717,z 506.764099,a -18.1002808,b -7.89086008,c -34.6327782,s 2,t 42,e1 0.0,e2 0.0,e3 0.0,e4 0.0,e5 0.0,e6 0.0}
DECL FDAT Fp1307={TOOL_NO 1,BASE_NO 2,IPO_FRAME #BASE}
DECL PDAT PPDAT132={VEL 100.0,ACC 85.0,APO_DIST 100.0}
DECL SPOT_SUGG_T LAST_SPOT={GUN[] " 1                      ",RETR_CMD[] "#OPN                    ",CHOISE[] "#FIRST                  ",CLO_TM[] "1                       ",PGNO1[] " 1                      ",PRESS1[] "0                       ",PGNO2[] " 1                      ",PRESS2[] "0                       ",SPOT_PARAMS[] "NORMAL                  "}
DECL E6POS Xswp_60_0800={x 452.408905,y 900.328918,z 1036.31494,a 69.1045532,b -12.6671,c -63.8056107,s 2,t 43,e1 0.0,e2 0.0,e3 0.0,e4 0.0,e5 0.0,e6 0.0}
DECL FDAT Fswp_60_0800={TOOL_NO 1,BASE_NO 2,IPO_FRAME #BASE}
DECL E6POS Xswp_60_0780={x 261.927307,y 927.338501,z 668.966919,a 66.255661,b -11.8886003,c -62.0566101,s 2,t 43,e1 0.0,e2 0.0,e3 0.0,e4 0.0,e5 0.0,e6 0.0}
DECL FDAT Fswp_60_0780={TOOL_NO 1,BASE_NO 2,IPO_FRAME #BASE}
DECL E6POS XP1308={x 207.306396,y 885.891113,z 568.437805,a 81.2640228,b 16.4622803,c -61.4363785,s 2,t 43,e1 0.0,e2 0.0,e3 0.0,e4 0.0,e5 0.0,e6 0.0}
DECL FDAT Fp1308={TOOL_NO 1,BASE_NO 2,IPO_FRAME #BASE}
DECL PDAT PPDAT133={VEL 100.0,ACC 80.0,APO_DIST 100.0}
ENDDAT
